# B&R Automation Studio project 305841_E00002_AM_0
Automation Studio 4.11.2.75; technology packages: mapp 5.17.0, mappCockpit 5.17.0, mappControl 5.17.0, mappMotion 5.17.1, mappSafety 5.17.0, mappView 5.17.0

## Configuration EchCm_AM

### Task classes (Cpu.sw)
```
Cyclic#2 (cycle 6000 us, tolerance 6000 us):
  ProdCycle <- PlcLogic.ProdCycle.prg
  Annunc <- PlcLogic.Annunc.prg
Cyclic#3 (cycle 12000 us, tolerance 12000 us):
  Pendant <- PlcLogic.Pendant.prg
  ProcInputs <- PlcLogic.ProcInputs.prg
  axSpinSM <- PlcLogic.axSpindle.axSpindleSM.prg
  axOutESM <- PlcLogic.axOutE.axOutESM.prg
  axInESM <- PlcLogic.axInE.axInESM.prg
  axZSM <- PlcLogic.axZ.axZSM.prg
  axHwSM <- PlcLogic.axHandwheel.axHwSM.prg
  axCfVfdSM <- PlcLogic.axCfVfd.axCfVfdSM.prg
Cyclic#4 (cycle 48000 us, tolerance 48000 us):
  AxEnable <- PlcLogic.AxEnable.prg
  CuttingFlu <- PlcLogic.CuttingFluidVFD.prg
  OmSafeDev <- PlcLogic.OmSafeDev.prg
  DepthToAng <- PlcLogic.DepthLookup.DepthToAngle.prg
DataObjects: McAcpSys
NcDataObjects: axSpindleP <- PlcLogic.axSpindle.axSpindleParamTable.dob, axOutEPara <- PlcLogic.axOutE.axOutEParamTable.dob, axInEParam <- PlcLogic.axInE.axInEParamTable.dob, axZParamTa <- PlcLogic.axZ.axZParamTable.dob, Cam1P <- PlcLogic.axInE.Cam1P.dob, Cam1P_Fp <- PlcLogic.axInE.Cam1P_Fp.dob, Cam2P <- PlcLogic.axInE.Cam2P.dob, Cam2P_Fp <- PlcLogic.axInE.Cam2P_Fp.dob, Cam3P <- PlcLogic.axInE.Cam3P.dob, Cam3P_Fp <- PlcLogic.axInE.Cam3P_Fp.dob, Cam4P <- PlcLogic.axInE.Cam4P.dob, Cam4P_Fp <- PlcLogic.axInE.Cam4P_Fp.dob, Cam5P <- PlcLogic.axInE.Cam5P.dob, Cam5P_Fp <- PlcLogic.axInE.Cam5P_Fp.dob, Cam6P <- PlcLogic.axInE.Cam6P.dob, Cam6P_Fp <- PlcLogic.axInE.Cam6P_Fp.dob, McDriveLog
Binaries: udbdef, mvLoader, arflatprv, TCData, FWRules, arcoal, arsvcreg, McAcpSim, McProfGen, McAcpDrv, mCoWebSc, TCLang, OpcUaSrv, DataObject, Settings, iomap, asfw, axCfgZ, Role, ashwac, sysconf, arconfig, ashwd, Config, axCfgInE, axCfgSpin, asiol1, axCfgOutE, Anonymous, User, cockpit1, TC, vAxHwCfg, vAxHw, axCfgCfPmp, CamFeature, camlist1, mappConfig, vAxHwLin, vAxHwRot, wgRecipe, cmRecipe, HwLinCfg, Config_5, HwRotCfg, Config_3
Libraries: sys_lib, runtime, brsystem, GAProcIO, standard, McBase, SfDomain, MpAxis, McAxis, MpBase, MpRecipe, McAcpAx, GAMpMotion, McPureVAx, astime, AsBrStr, GAConvert, MpAlarmX, AsBrMath, GAMath, CoTrace, AsZip, FileIO, McDS402Ax, astcp, asieccon, asiodiag, asepl, SfDomDrv, asusb, SfDomVis, aruser, arssl, powerlnk, MpSfDomMgr, dataobj, asioacc, GAMotor, MTFilter, MTBasics, MTTypes
```

### Hardware
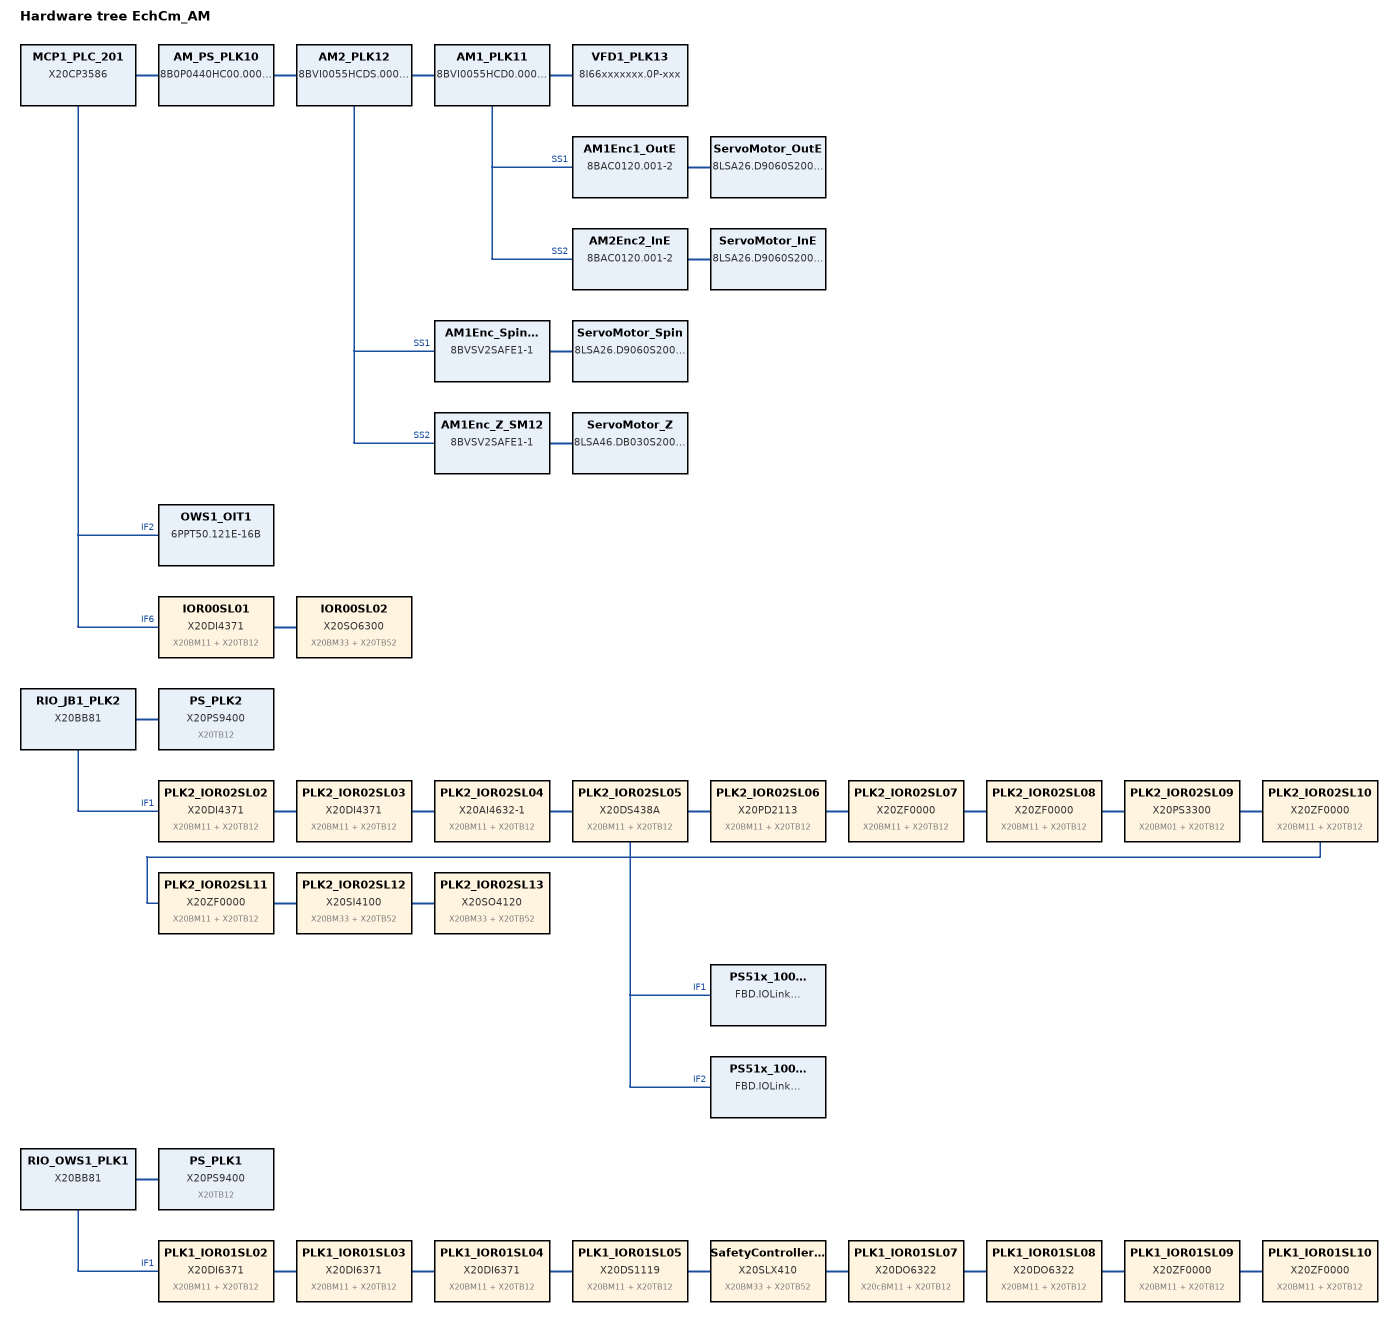
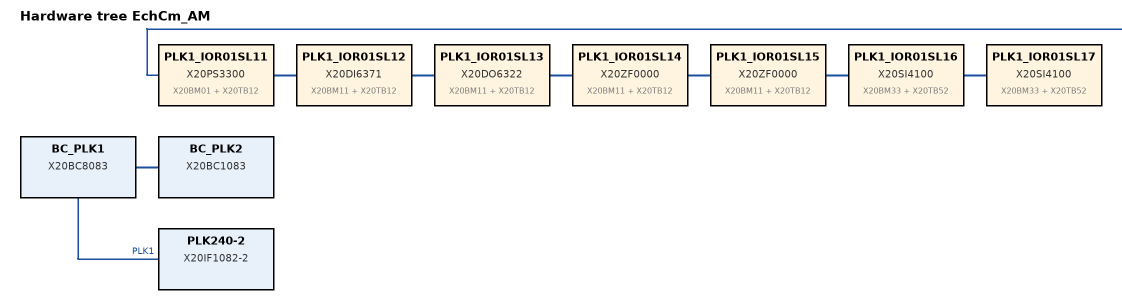
```
AM1Enc1_OutE : 8BAC0120.001-2 v2.2.0.0  [SS -> AM1_PLK11.SS1]
  PlugInType = Encoder
  McAcoposTypeID = AcoposMultiPlugInConfig
AM1Enc_Spin_SM11 : 8BVSV2SAFE1-1 v2.2.0.0  [SS -> AM2_PLK12.SS1]
  SafeModuleID = 11
  PlugInType = Encoder
  McAcoposTypeID = AcoposMultiPlugInConfig
AM1Enc_Z_SM12 : 8BVSV2SAFE1-1 v2.2.0.0  [SS -> AM2_PLK12.SS2]
  SafeModuleID = 12
  PlugInType = Encoder
  McAcoposTypeID = AcoposMultiPlugInConfig
AM1_PLK11 : 8BVI0055HCD0.000-1 v2.3.0.1  [PLK1 -> AM2_PLK12.PLK2 (NodeNumber=11) [Cable Type=PowerlinkCable, Length=10, Version=1.0.0.3]; PLK2 -> VFD1_PLK13.PLK1 (NodeNumber=11) [Cable Type=PowerlinkCable, Length=10, Version=1.0.0.3]; MT2 -> ServoMotor_InE.MT]
  DriveConfiguration/Module:
    McAcoposTypeID = AcoposP3SConfig
    ActivateACOPOSSimulationOnPLC = 0
  DriveConfiguration/Module/PowerSupply:
    PowerSupplyModuleReference = AM_PS
  DriveConfiguration/Channel[1]/RealAxis:
    AxisReference = gAxOutE
    MechanicalElementsIsInvisible = 0
  DriveConfiguration/Channel[1]/RealAxis/MechanicalElements/Gearbox:
    InputIsReadOnly = 0
    Input = 25
    OutputIsReadOnly = 0
    Output = 1
  DriveConfiguration/Channel[1]/RealAxis/MechanicalElements/RotaryToLinearTransformation:
    ReferenceDistanceIsReadOnly = 0
    ReferenceDistance = 360.0
  DriveConfiguration/Channel[1]/RealAxis/Controller:
    ModeIsReadOnly = 0
    Mode = PositionController
  DriveConfiguration/Channel[1]/RealAxis/Controller/Mode/Position:
    ProportionalGain = 462
    IntegrationTime = 0.0
    PredictionTime = 0.0004
    TotalDelayTime = 0.0004
  DriveConfiguration/Channel[1]/RealAxis/Controller/Mode/Speed:
    ProportionalGainIsReadOnly = 0
    ProportionalGain = 0.35
    IntegrationTimeIsReadOnly = 0
    IntegrationTime = 0.0
    FilterTimeIsReadOnly = 0
    FilterTime = 0.0
  DriveConfiguration/Channel[1]/RealAxis/Controller/Mode/LoopFilters:
    LoopFilterXIsReadOnly = 0
    LoopFilter1 = NotUsed
    LoopFilter2 = NotUsed
    LoopFilter3 = NotUsed
  DriveConfiguration/Channel[1]/RealAxis/Homing:
    ModeIsReadOnly = 0
    Mode = RestorePosition
    RestorePositionVariable = ::gr_AxOutERestorePos
  DriveConfiguration/Channel[1]/RealAxis/StopReaction:
    QuickstopIsReadOnly = 0
    Quickstop = DecelerationLimit
    DriveErrorIsReadOnly = 0
    DriveError = DecelerationLimit
  DriveConfiguration/Channel[1]/RealAxis/MovementErrorLimits:
    PositionError = 1.0
    VelocityErrorMonitoring = Automatic1
  DriveConfiguration/Channel[1]/RealAxis:
    JerkFilterIsReadOnly = 0
    JerkFilter = NotUsed
  DriveConfiguration/Channel[1]/RealAxis/DigitalInputs/HomingSwitch:
    SourceIsReadOnly = 0
    Source = NotUsed
    Level = High
  DriveConfiguration/Channel[1]/RealAxis/DigitalInputs/PositiveLimitSwitch:
    SourceIsReadOnly = 0
    Source = NotUsed
    Level = High
  DriveConfiguration/Channel[1]/RealAxis/DigitalInputs/NegativeLimitSwitch:
    SourceIsReadOnly = 0
    Source = NotUsed
    Level = High
  DriveConfiguration/Channel[1]/RealAxis/DigitalInputs/Trigger1:
    Source = X2Trigger1
    Level = High
  DriveConfiguration/Channel[1]/RealAxis/DigitalInputs/Trigger2:
    Source = X2Trigger2
    Level = High
  DriveConfiguration/Channel[1]/RealAxis/DigitalInputs/Quickstop:
    Input = NotUsed
  DriveConfiguration/Channel[1]/RealAxis/Simulation:
    SimulationModeOnPLC = SetValueGeneration
    SimulationModeOnACOPOS = NotUsed
  DriveConfiguration/Channel[1]:
    ExternalEncoderAxis = NotUsed
  DriveConfiguration/Channel[2]/RealAxis:
    AxisReference = gAxInE
    MechanicalElementsIsInvisible = 0
  DriveConfiguration/Channel[2]/RealAxis/MechanicalElements/Gearbox:
    InputIsReadOnly = 0
    Input = 25
    OutputIsReadOnly = 0
    Output = 1
  DriveConfiguration/Channel[2]/RealAxis/MechanicalElements/RotaryToLinearTransformation:
    ReferenceDistanceIsReadOnly = 0
    ReferenceDistance = 360.0
  DriveConfiguration/Channel[2]/RealAxis/Controller:
    ModeIsReadOnly = 0
    Mode = PositionController
  DriveConfiguration/Channel[2]/RealAxis/Controller/Mode/Position:
    ProportionalGain = 451.5
    IntegrationTime = 0.0
    PredictionTime = 0.0004
    TotalDelayTime = 0.0004
  DriveConfiguration/Channel[2]/RealAxis/Controller/Mode/Speed:
    ProportionalGainIsReadOnly = 0
    ProportionalGain = 0.325
    IntegrationTimeIsReadOnly = 0
    IntegrationTime = 0.0
    FilterTimeIsReadOnly = 0
    FilterTime = 0.0
  DriveConfiguration/Channel[2]/RealAxis/Controller/Mode/LoopFilters:
    LoopFilterXIsReadOnly = 0
    LoopFilter1 = NotUsed
    LoopFilter2 = NotUsed
    LoopFilter3 = NotUsed
  DriveConfiguration/Channel[2]/RealAxis/Homing:
    ModeIsReadOnly = 0
    Mode = RestorePosition
    RestorePositionVariable = ::gr_AxInERestorePos
  DriveConfiguration/Channel[2]/RealAxis/StopReaction:
    QuickstopIsReadOnly = 0
    Quickstop = DecelerationLimit
    DriveErrorIsReadOnly = 0
    DriveError = DecelerationLimit
  DriveConfiguration/Channel[2]/RealAxis/MovementErrorLimits:
    PositionError = 0.9
    VelocityErrorMonitoring = Automatic1
  DriveConfiguration/Channel[2]/RealAxis:
    JerkFilterIsReadOnly = 0
    JerkFilter = NotUsed
  DriveConfiguration/Channel[2]/RealAxis/DigitalInputs/HomingSwitch:
    SourceIsReadOnly = 0
    Source = NotUsed
    Level = High
  DriveConfiguration/Channel[2]/RealAxis/DigitalInputs/PositiveLimitSwitch:
    SourceIsReadOnly = 0
    Source = NotUsed
    Level = Low
  DriveConfiguration/Channel[2]/RealAxis/DigitalInputs/NegativeLimitSwitch:
    SourceIsReadOnly = 0
    Source = NotUsed
    Level = Low
  DriveConfiguration/Channel[2]/RealAxis/DigitalInputs/Trigger1:
    Source = X2Trigger1
    Level = High
  DriveConfiguration/Channel[2]/RealAxis/DigitalInputs/Trigger2:
    Source = X2Trigger2
    Level = High
  DriveConfiguration/Channel[2]/RealAxis/DigitalInputs/Quickstop:
    Input = NotUsed
  DriveConfiguration/Channel[2]/RealAxis/Simulation:
    SimulationModeOnPLC = SetValueGeneration
    SimulationModeOnACOPOS = NotUsed
  DriveConfiguration/Channel[2]/RealAxis/AxisFeatures:
    FeatureRef[1] = 
  DriveConfiguration/Channel[2]:
    ExternalEncoderAxis = NotUsed
  DriveConfiguration/Channel[2]/ChannelFeatures:
    FeatureRef[1] = Feature_CamList
AM2Enc2_InE : 8BAC0120.001-2 v2.2.0.0  [SS -> AM1_PLK11.SS2]
  PlugInType = Encoder
  McAcoposTypeID = AcoposMultiPlugInConfig
AM2_PLK12 : 8BVI0055HCDS.000-1 v2.3.0.1  [PLK1 -> AM_PS_PLK10.PLK2 (NodeNumber=12) [Cable Type=PowerlinkCable, Length=10, Version=1.0.0.3]; PLK2 -> AM1_PLK11.PLK1 (NodeNumber=12) [Cable Type=PowerlinkCable, Length=10, Version=1.0.0.3]; MT2 -> ServoMotor_Z.MT]
  DriveConfiguration/Module:
    McAcoposTypeID = AcoposMultiDConfig
    ActivateACOPOSSimulationOnPLC = 0
  DriveConfiguration/Module/PowerSupply:
    PowerSupplyModuleReference = AM_PS
  DriveConfiguration/Channel[1]/RealAxis:
    AxisReference = gAxSpin
    MechanicalElementsIsInvisible = 0
  DriveConfiguration/Channel[1]/RealAxis/MechanicalElements/Gearbox:
    InputIsReadOnly = 0
    Input = 10
    OutputIsReadOnly = 0
    Output = 1
  DriveConfiguration/Channel[1]/RealAxis/MechanicalElements/RotaryToLinearTransformation:
    ReferenceDistanceIsReadOnly = 0
    ReferenceDistance = 1
  DriveConfiguration/Channel[1]/RealAxis/Controller:
    ModeIsReadOnly = 0
    Mode = PositionController
  DriveConfiguration/Channel[1]/RealAxis/Controller/Mode/Position:
    ProportionalGain = 526
    IntegrationTime = 0.0
    PredictionTime = 0.0004
    TotalDelayTime = 0.0004
  DriveConfiguration/Channel[1]/RealAxis/Controller/Mode/Speed:
    ProportionalGainIsReadOnly = 0
    ProportionalGain = 0.25
    IntegrationTimeIsReadOnly = 0
    IntegrationTime = 0
    FilterTimeIsReadOnly = 0
    FilterTime = 0
  DriveConfiguration/Channel[1]/RealAxis/Controller/Mode/LoopFilters:
    LoopFilterXIsReadOnly = 0
    LoopFilter1 = NotUsed
    LoopFilter2 = NotUsed
    LoopFilter3 = NotUsed
  DriveConfiguration/Channel[1]/RealAxis/Homing:
    ModeIsReadOnly = 0
    Mode = RestorePosition
    RestorePositionVariable = ::gr_AxSpinRestorePos
  DriveConfiguration/Channel[1]/RealAxis/StopReaction:
    QuickstopIsReadOnly = 0
    Quickstop = DecelerationLimit
    DriveErrorIsReadOnly = 0
    DriveError = DecelerationLimit
  DriveConfiguration/Channel[1]/RealAxis/MovementErrorLimits:
    PositionError = 1.0
    VelocityErrorMonitoring = Automatic1
  DriveConfiguration/Channel[1]/RealAxis:
    JerkFilterIsReadOnly = 0
    JerkFilter = NotUsed
  DriveConfiguration/Channel[1]/RealAxis/DigitalInputs/HomingSwitch:
    SourceIsReadOnly = 0
    Source = NotUsed
    Level = High
  DriveConfiguration/Channel[1]/RealAxis/DigitalInputs/PositiveLimitSwitch:
    SourceIsReadOnly = 0
    Source = NotUsed
    Level = High
  DriveConfiguration/Channel[1]/RealAxis/DigitalInputs/NegativeLimitSwitch:
    SourceIsReadOnly = 0
    Source = NotUsed
    Level = High
  DriveConfiguration/Channel[1]/RealAxis/DigitalInputs/Trigger1:
    Source = X2Trigger1
    Level = High
  DriveConfiguration/Channel[1]/RealAxis/DigitalInputs/Trigger2:
    Source = X2Trigger2
    Level = High
  DriveConfiguration/Channel[1]/RealAxis/DigitalInputs/Quickstop:
    Input = NotUsed
  DriveConfiguration/Channel[1]/RealAxis/Simulation:
    SimulationModeOnPLC = SetValueGeneration
    SimulationModeOnACOPOS = NotUsed
  DriveConfiguration/Channel[1]:
    ExternalEncoderAxis = NotUsed
  DriveConfiguration/Channel[2]/RealAxis:
    AxisReference = gAxZ
    MechanicalElementsIsInvisible = 0
  DriveConfiguration/Channel[2]/RealAxis/MechanicalElements/Gearbox:
    InputIsReadOnly = 0
    Input = 1
    OutputIsReadOnly = 0
    Output = 1
  DriveConfiguration/Channel[2]/RealAxis/MechanicalElements/RotaryToLinearTransformation:
    ReferenceDistanceIsReadOnly = 0
    ReferenceDistance = 5.08
  DriveConfiguration/Channel[2]/RealAxis/Controller:
    ModeIsReadOnly = 0
    Mode = PositionController
  DriveConfiguration/Channel[2]/RealAxis/Controller/Mode/Position:
    ProportionalGain = 551
    IntegrationTime = 0.0
    PredictionTime = 0.0004
    TotalDelayTime = 0.0004
  DriveConfiguration/Channel[2]/RealAxis/Controller/Mode/Speed:
    ProportionalGainIsReadOnly = 0
    ProportionalGain = 1.0
    IntegrationTimeIsReadOnly = 0
    IntegrationTime = 0.0
    FilterTimeIsReadOnly = 0
    FilterTime = 0.0
  DriveConfiguration/Channel[2]/RealAxis/Controller/Mode/LoopFilters:
    LoopFilterXIsReadOnly = 0
    LoopFilter1 = NotUsed
    LoopFilter2 = NotUsed
    LoopFilter3 = NotUsed
  DriveConfiguration/Channel[2]/RealAxis/Homing:
    ModeIsReadOnly = 0
    Mode = RestorePosition
    RestorePositionVariable = ::gr_AxZRestorePos
  DriveConfiguration/Channel[2]/RealAxis/StopReaction:
    QuickstopIsReadOnly = 0
    Quickstop = DecelerationLimit
    DriveErrorIsReadOnly = 0
    DriveError = DecelerationLimit
  DriveConfiguration/Channel[2]/RealAxis/MovementErrorLimits:
    PositionError = 1.0
    VelocityErrorMonitoring = Automatic1
  DriveConfiguration/Channel[2]/RealAxis:
    JerkFilterIsReadOnly = 0
    JerkFilter = NotUsed
  DriveConfiguration/Channel[2]/RealAxis/DigitalInputs/HomingSwitch:
    SourceIsReadOnly = 0
    Source = NotUsed
    Level = High
  DriveConfiguration/Channel[2]/RealAxis/DigitalInputs/PositiveLimitSwitch:
    SourceIsReadOnly = 0
    Source = X2Trigger1
    Level = Low
  DriveConfiguration/Channel[2]/RealAxis/DigitalInputs/NegativeLimitSwitch:
    SourceIsReadOnly = 0
    Source = X2Trigger2
    Level = Low
  DriveConfiguration/Channel[2]/RealAxis/DigitalInputs/Trigger1:
    Source = X2Trigger1
    Level = High
  DriveConfiguration/Channel[2]/RealAxis/DigitalInputs/Trigger2:
    Source = X2Trigger2
    Level = High
  DriveConfiguration/Channel[2]/RealAxis/DigitalInputs/Quickstop:
    Input = NotUsed
  DriveConfiguration/Channel[2]/RealAxis/Simulation:
    SimulationModeOnPLC = SetValueGeneration
    SimulationModeOnACOPOS = NotUsed
  DriveConfiguration/Channel[2]/RealAxis/AxisFeatures:
    FeatureRef[1] = 
  DriveConfiguration/Channel[2]:
    ExternalEncoderAxis = NotUsed
AM_PS_PLK10 : 8B0P0440HC00.000-1 v2.3.0.1  [PLK1 -> MCP1_PLC_201.IF3 (NodeNumber=10) [Cable Type=PowerlinkCable, Length=10, Version=1.0.0.3]; PLK2 -> AM2_PLK12.PLK1 (NodeNumber=10) [Cable Type=PowerlinkCable, Length=10, Version=1.0.0.3]]
  DriveConfiguration/Module:
    McAcoposTypeID = AcoposMultiPSMpConfig
    ActivateACOPOSSimulationOnPLC = 0
  DriveConfiguration/Channel[1]/PowerSection:
    AxisReference = AM_PS
BC_PLK1 : X20BC8083 v2.14.0.0  [PLK1 -> PLK240-2.PLK2 (NodeNumber=1) [Cable Type=PowerlinkCable, Length=10, Version=1.0.0.3]; PLK2 -> BC_PLK2.PLK1 (NodeNumber=1) [Cable Type=PowerlinkCable, Length=10, Version=1.0.0.3]; SL -> RIO_OWS1_PLK1.SL1]
BC_PLK2 : X20BC1083 v2.14.0.0  [PLK1 -> BC_PLK1.PLK2 (NodeNumber=2) [Cable Type=PowerlinkCable, Length=10, Version=1.0.0.3]; SL -> RIO_JB1_PLK2.SL1]
IOR00SL01 : X20DI4371 v1.2.0.0  [SS1 -> X20TB12.SS; SL -> X20BM11.SL1]
IOR00SL02 : X20SO6300 v2.3.0.0  [SS1 -> X20TB52d.SS; SL -> X20BM33d.SL1]
  DigitalOutput01 = viaSafeLOGIC
  DigitalOutput02 = viaSafeLOGIC
  DigitalOutput03 = viaSafeLOGIC
  DigitalOutput04 = viaSafeLOGIC
  DigitalOutput05 = viaSafeLOGIC
  DigitalOutput06 = viaSafeLOGIC
MCP1_PLC_201 : X20CP3586 v1.10.0.0
  Connector IF2:
    ActivateDevice = 1
    HostName = plc_mcp1
    Mode = Manual
    InternetAddress = 10.10.2.240
    SubnetMask = 255.255.255.0
  Connector IF3:
    EplHostName = PLC_MCP1_PLK1
    CycleTime = 800
  ConfigurationID = 305841_E00002_Rev0_PLC_Main
  ConfigVersion = 0.0.0
  UserPartitionSize = 20
  AutomaticTransferOfUserfiles = on
  PermanentPvSize = 9216
  VolatileGlobalPvSize = 69630
  CyclicTaskClassCount = 6
  Cyclic1Duration = 2000
  Cyclic1Tolerance = 2000
  Cyclic2Duration = 6000
  Cyclic2Tolerance = 6000
  Cyclic3Duration = 12000
  Cyclic3Tolerance = 12000
  Cyclic4Duration = 48000
  Cyclic4Tolerance = 48000
  Cyclic5Duration = 96000
  Cyclic5Tolerance = 9600000
  Cyclic6Duration = 480000
  Cyclic6Tolerance = 480000
  FileDevice1
  FileDeviceName1 = UserPartitionRoot
  FileDevicePath1 = F:\
  FileDevice2
  FileDeviceName2 = Recipes
  FileDevicePath2 = F:\config\recipes\
  FileDevice3
  FileDeviceName3 = IOConfig
  FileDevicePath3 = F:\config\io\
  EthernetHostName = mcp1_plc201
  FtpUser1
  FtpUsername1 = ftpuser
  FtpUserPassword1 = wzi3iB5UNI3uCms7ZCmB0Woh2QaOICjzuPm+LM5DkNg=
  FtpUserSalt1 = UFkRbDjT
  FTPAccessRight1 = 0
  ActivateOpcUa = 1
  OpcUaPort = 4841
  OpcUaInformationModels_PV_Version = 1
OWS1_OIT1 : 6PPT50.121E-16B v1.3.8.0  [ETH1 -> MCP1_PLC_201.IF2 [Cable Type=PowerlinkCable, Length=10, Version=1.0.0.3]]
  Terminal = true
  Mode = Manual
  InternetAddress = 10.10.2.20
  Subnetmask = 255.255.255.0
  Hostname = ows1_oit1
  PasswordVNC = 
  PasswordCIFS = 
  PasswordService = 
PLK1_IOR01SL02 : X20DI6371 v1.2.0.0  [SS1 -> X20TB12n.SS; SL -> X20BM11l.SL1]
  InputFilter = 250
PLK1_IOR01SL03 : X20DI6371 v1.2.0.0  [SS1 -> X20TB12c.SS; SL -> X20BM11c.SL1]
  InputFilter = 250
PLK1_IOR01SL04 : X20DI6371 v1.2.0.0  [SS1 -> X20TB12ab.SS; SL -> X20BM11x.SL1]
  InputFilter = 250
PLK1_IOR01SL05 : X20DS1119 v1.5.0.0  [SS1 -> X20TB12e.SS; SL -> X20BM11e.SL1]
  PSInfo = on
  SDCInfo = on
  NetworkInfo = 8Bit
  Function03 = AB
PLK1_IOR01SL07 : X20DO6322 v1.3.0.0  [SS1 -> X20TB12p.SS; SL -> X20cBM11a.SL1]
PLK1_IOR01SL08 : X20DO6322 v1.3.0.0  [SS1 -> X20TB12h.SS; SL -> X20BM11h.SL1]
PLK1_IOR01SL09 : X20ZF0000 v1.1.0.0 (Disabled=true)  [SS1 -> X20TB12o.SS; SL -> X20BM11n.SL1]
PLK1_IOR01SL10 : X20ZF0000 v1.1.0.0 (Disabled=true)  [SS1 -> X20TB12i.SS; SL -> X20BM11m.SL1]
PLK1_IOR01SL11 : X20PS3300 v1.4.0.0  [SS1 -> X20TB12z.SS; SL -> X20BM01.SL1]
  PowerInfo = on
PLK1_IOR01SL12 : X20DI6371 v1.2.0.0  [SS1 -> X20TB12d.SS; SL -> X20BM11d.SL1]
PLK1_IOR01SL13 : X20DO6322 v1.3.0.0  [SS1 -> X20TB12b.SS; SL -> X20BM11b.SL1]
  Supervision = off
PLK1_IOR01SL14 : X20ZF0000 v1.1.0.0 (Disabled=true)  [SS1 -> X20TB12f.SS; SL -> X20BM11f.SL1]
PLK1_IOR01SL15 : X20ZF0000 v1.1.0.0 (Disabled=true)  [SS1 -> X20TB12q.SS; SL -> X20BM11o.SL1]
PLK1_IOR01SL16 : X20SI4100 v2.4.0.0  [SS1 -> X20TB52b.SS; SL -> X20BM33b.SL1]
  SafeModuleID = 116
PLK1_IOR01SL17 : X20SI4100 v2.4.0.0  [SS1 -> X20TB52a.SS; SL -> X20BM33a.SL1]
  SafeModuleID = 117
PLK240-2 : X20IF1082-2 v1.14.0.0  [PLK2 -> BC_PLK1.PLK1 [Cable Type=PowerlinkCable, Length=10, Version=1.0.0.3]; SS -> MCP1_PLC_201.SS1]
  Connector IF1:
    EplHostName = PLC_MCP1_PLK2
    NodeDefinition = Software
    EplNatSubnet = 192.168.102.0
PLK2_IOR02SL02 : X20DI4371 v1.2.0.0  [SS1 -> X20TB12s.SS; SL -> X20BM11p.SL1]
PLK2_IOR02SL03 : X20DI4371 v1.2.0.0  [SS1 -> X20TB12t.SS; SL -> X20BM11q.SL1]
PLK2_IOR02SL04 : X20AI4632-1 v1.2.0.0  [SS1 -> X20TB12u.SS; SL -> X20BM11r.SL1]
  ChannelType01 = 0 to 22mA
  ChannelType02 = 0 to 22mA
  Channel03enable = off
  Channel04enable = off
PLK2_IOR02SL05 : X20DS438A v2.4.0.0  [SS1 -> X20TB12aa.SS; SL -> X20BM11w.SL1]
  DtmRef = FBD.BRIOLinkModuleDTM.DTMCore.X20DS438A
  DtmId = 7db43003-0ff5-4bbd-8923-86eacecae911
  CommDtmId = ab9d1316-8c35-4493-ab34-f7b1b8ca9169
  RequiresDTMBuild = true
  ConfigFile = Communication.dtm
  ConfigModule = asiol1
  OperatingMode01 = Operate
  PDI_Enable01 = variousTypes
  PDI_DataType01_1 = UINT
  OperatingMode02 = Operate
  PDI_Enable02 = variousTypes
  PDI_DataType02_1 = UINT
PLK2_IOR02SL06 : X20PD2113 v1.2.0.0  [SS1 -> X20TB12g.SS; SL -> X20BM11g.SL1]
PLK2_IOR02SL07 : X20ZF0000 v1.1.0.0 (Disabled=true)  [SS1 -> X20TB12x.SS; SL -> X20BM11t.SL1]
PLK2_IOR02SL08 : X20ZF0000 v1.1.0.0 (Disabled=true)  [SS1 -> X20TB12w.SS; SL -> X20BM11v.SL1]
PLK2_IOR02SL09 : X20PS3300 v1.4.0.0 (Disabled=true)  [SS1 -> X20TB12ac.SS; SL -> X20BM01a.SL1]
  PowerInfo = on
PLK2_IOR02SL10 : X20ZF0000 v1.1.0.0 (Disabled=true)  [SS1 -> X20TB12y.SS; SL -> X20BM11u.SL1]
PLK2_IOR02SL11 : X20ZF0000 v1.1.0.0 (Disabled=true)  [SS1 -> X20TB12v.SS; SL -> X20BM11s.SL1]
PLK2_IOR02SL12 : X20SI4100 v2.4.0.0  [SS1 -> X20TB52c.SS; SL -> X20BM33c.SL1]
  SafeModuleID = 212
PLK2_IOR02SL13 : X20SO4120 v2.3.0.0  [SS1 -> X20TB52e.SS; SL -> X20BM33e.SL1]
  PLCopenInfo = on
  SafeModuleID = 213
  DigitalOutput01 = viaSafeLOGIC
  DigitalOutput02 = viaSafeLOGIC
  DigitalOutput03 = viaSafeLOGIC
  DigitalOutput04 = viaSafeLOGIC
PS51x_100_LI2UPN8_IODD1_1 : FBD.IOLink.GenericDeviceDTM.DTMCore.PS51x-100-LI2UPN8 IODD1.1 v2.9 (OrderNumber=PS51x-100-LI2UPN8 IODD1.1)  [IO-Link1 -> PLK2_IOR02SL05.IF1]
  DtmId = 9f03f336-de2c-4174-a814-ce0739b6707c
PS51x_100_LI2UPN8_IODD1_1a : FBD.IOLink.GenericDeviceDTM.DTMCore.PS51x-100-LI2UPN8 IODD1.1 v2.9 (OrderNumber=PS51x-100-LI2UPN8 IODD1.1)  [IO-Link1 -> PLK2_IOR02SL05.IF2]
  DtmId = 948ae1a5-f93f-40dc-8e06-a46fa964d649
PS_PLK1 : X20PS9400 v1.8.0.0  [SS1 -> X20TB12m.SS; PS -> RIO_OWS1_PLK1.PS1]
  PowerInfo = on
PS_PLK2 : X20PS9400 v1.8.0.0  [SS1 -> X20TB12r.SS; PS -> RIO_JB1_PLK2.PS1]
RIO_JB1_PLK2 : X20BB81 v1.1.0.0
RIO_OWS1_PLK1 : X20BB81 v1.1.0.0
SafetyController_R01SL06 : X20SLX410 v2.4.1.1  [SS1 -> X20TB52.SS; SL -> X20BM33.SL1]
  UnsafeOutputBOOLs = 24
  UnsafeInputBOOLs = 24
  UnsafeInputUINTs = 4
ServoMotor_InE : 8LSA26.D9060S200-3 v2.2.0.1  [EC -> AM2Enc2_InE.EC; MT -> AM1_PLK11.MT2]
  M1/MotorParameters:
    MOTOR_AMB_TEMP_RATED = 40
ServoMotor_OutE : 8LSA26.D9060S200-3 v2.2.0.1  [EC -> AM1Enc1_OutE.EC; MT -> AM1_PLK11.MT1]
  M1/MotorParameters:
    MOTOR_AMB_TEMP_RATED = 40
ServoMotor_Spin : 8LSA26.D9060S200-3 v2.2.0.1  [EC -> AM1Enc_Spin_SM11.EC; MT -> AM2_PLK12.MT1]
  M1/MotorParameters:
    MOTOR_AMB_TEMP_RATED = 40
ServoMotor_Z : 8LSA46.DB030S200-3 v2.2.0.1  [EC -> AM1Enc_Z_SM12.EC; MT -> AM2_PLK12.MT2]
  M1/MotorParameters:
    MOTOR_AMB_TEMP_RATED = 40
VFD1_PLK13 : 8I66xxxxxxx.0P-xxx v2.5.1.0  [PLK1 -> AM1_PLK11.PLK2 (NodeNumber=13) [Cable Type=PowerlinkCable, Length=10, Version=1.0.0.3]]
  Supervision = off
  PlkDiagnosisAdd = on
  FunctionModel = MotionConfig
  McTypeID = McAcoposInverterP66P
  AxisReference = gAxCfPmp
  InputIsReadOnly = 0
  Input = 1
  OutputIsReadOnly = 0
  Output = 1
  ReferenceDistanceIsReadOnly = 0
  ReferenceDistance = 1
  UnitOfSetpoint = Rpm
  IOM_AIDP1 = HMIS
  IOM_AIDP2 = LFT
  IOM_AIDP3 = ETAD_u
  Mode_LI3 = Safety
  Sel_NameplateMask = 8Ix6T401100_IEC
  Cfg_NSP = 1175
  Cfg_FRS = 600
  Cfg_UNS = 480
  Cfg_COS = 73
X20BM01 : X20BM01 v2.1.0.0  [X2X1 -> X20BM11m.X2X2]
X20BM01a : X20BM01 v2.1.0.0 (Disabled=true)  [X2X1 -> X20BM11v.X2X2]
X20BM11 : X20BM11 v1.1.0.0  [X2X1 -> MCP1_PLC_201.IF6]
X20BM11b : X20BM11 v1.1.0.0  [X2X1 -> X20BM11d.X2X2]
X20BM11c : X20BM11 v1.1.0.0  [X2X1 -> X20BM11l.X2X2]
X20BM11d : X20BM11 v1.1.0.0  [X2X1 -> X20BM01.X2X2]
X20BM11e : X20BM11 v1.1.0.0  [X2X1 -> X20BM11x.X2X2]
X20BM11f : X20BM11 v1.1.0.0 (Disabled=true)  [X2X1 -> X20BM11b.X2X2]
X20BM11g : X20BM11 v1.1.0.0  [X2X1 -> X20BM11w.X2X2]
X20BM11h : X20BM11 v1.1.0.0  [X2X1 -> X20cBM11a.X2X2]
X20BM11l : X20BM11 v1.1.0.0  [X2X1 -> RIO_OWS1_PLK1.IF1]
X20BM11m : X20BM11 v1.1.0.0 (Disabled=true)  [X2X1 -> X20BM11n.X2X2]
X20BM11n : X20BM11 v1.1.0.0 (Disabled=true)  [X2X1 -> X20BM11h.X2X2]
X20BM11o : X20BM11 v1.1.0.0 (Disabled=true)  [X2X1 -> X20BM11f.X2X2]
X20BM11p : X20BM11 v1.1.0.0  [X2X1 -> RIO_JB1_PLK2.IF1]
X20BM11q : X20BM11 v1.1.0.0  [X2X1 -> X20BM11p.X2X2]
X20BM11r : X20BM11 v1.1.0.0  [X2X1 -> X20BM11q.X2X2]
X20BM11s : X20BM11 v1.1.0.0 (Disabled=true)  [X2X1 -> X20BM11u.X2X2]
X20BM11t : X20BM11 v1.1.0.0 (Disabled=true)  [X2X1 -> X20BM11g.X2X2]
X20BM11u : X20BM11 v1.1.0.0 (Disabled=true)  [X2X1 -> X20BM01a.X2X2]
X20BM11v : X20BM11 v1.1.0.0 (Disabled=true)  [X2X1 -> X20BM11t.X2X2]
X20BM11w : X20BM11 v1.1.0.0  [X2X1 -> X20BM11r.X2X2]
X20BM11x : X20BM11 v1.1.0.0  [X2X1 -> X20BM11c.X2X2]
X20BM33 : X20BM33 v1.0.0.6  [X2X1 -> X20BM11e.X2X2]
X20BM33a : X20BM33 v1.0.0.6  [X2X1 -> X20BM33b.X2X2]
X20BM33b : X20BM33 v1.0.0.6  [X2X1 -> X20BM11o.X2X2]
X20BM33c : X20BM33 v1.0.0.6  [X2X1 -> X20BM11s.X2X2]
X20BM33d : X20BM33 v1.0.0.6  [X2X1 -> X20BM11.X2X2]
X20BM33e : X20BM33 v1.0.0.6  [X2X1 -> X20BM33c.X2X2]
X20TB12 : X20TB12 v1.0.0.0
X20TB12aa : X20TB12 v1.0.0.0
X20TB12ab : X20TB12 v1.0.0.0
X20TB12ac : X20TB12 v1.0.0.0 (Disabled=true)
X20TB12b : X20TB12 v1.0.0.0
X20TB12c : X20TB12 v1.0.0.0
X20TB12d : X20TB12 v1.0.0.0
X20TB12e : X20TB12 v1.0.0.0
X20TB12f : X20TB12 v1.0.0.0 (Disabled=true)
X20TB12g : X20TB12 v1.0.0.0
X20TB12h : X20TB12 v1.0.0.0
X20TB12i : X20TB12 v1.0.0.0 (Disabled=true)
X20TB12m : X20TB12 v1.0.0.0
X20TB12n : X20TB12 v1.0.0.0
X20TB12o : X20TB12 v1.0.0.0 (Disabled=true)
X20TB12p : X20TB12 v1.0.0.0
X20TB12q : X20TB12 v1.0.0.0 (Disabled=true)
X20TB12r : X20TB12 v1.0.0.0
X20TB12s : X20TB12 v1.0.0.0
X20TB12t : X20TB12 v1.0.0.0
X20TB12u : X20TB12 v1.0.0.0
X20TB12v : X20TB12 v1.0.0.0 (Disabled=true)
X20TB12w : X20TB12 v1.0.0.0 (Disabled=true)
X20TB12x : X20TB12 v1.0.0.0 (Disabled=true)
X20TB12y : X20TB12 v1.0.0.0 (Disabled=true)
X20TB12z : X20TB12 v1.0.0.0
X20TB52 : X20TB52 v1.0.0.2
X20TB52a : X20TB52 v1.0.0.2
X20TB52b : X20TB52 v1.0.0.2
X20TB52c : X20TB52 v1.0.0.2
X20TB52d : X20TB52 v1.0.0.2
X20TB52e : X20TB52 v1.0.0.2
X20cBM11a : X20cBM11 v1.0.1.0  [X2X1 -> X20BM33.X2X2]
```

### Cpu.per - MCP1_PLC_201/Cpu.per
```iecst
VAR_CONFIG
	gr_AxSpindleRestorePos AT %M0; (* *)
	gr_AxOutERestorePos AT %M72; (* *)
	gr_AxInERestorePos AT %M144; (* *)
	gr_AxZRestorePos AT %M216; (* *)
	gr_AI_FT_CFFlow_Params AT %M288; (* *)
	gr_AI_LT_CFTankLevel_Params AT %M376; (* *)
	gr_AI_PT_CFFilterOutlet_Params AT %M464; (* *)
	gr_AI_PT_CFPumpOutlet_Params AT %M552; (* *)
	gr_AI_DP_CFFilter_Params AT %M640; (* *)
	gr_DI_JI_480VACOk_Params AT %M728; (* *)
	gr_DI_LSL_CFTank_Params AT %M760; (* *)
	gr_DI_ZS_CFTankLocator_Params AT %M792; (* *)
	gr_AxisPositionLimits AT %M824; (* *)
	gr_CfgCurrent AT %M968; (* *)
	gr_PartCurrent AT %M1152; (* *)
END_VAR
```

### IoMap.iom - MCP1_PLC_201/IoMap.iom
```iecst
VAR_CONFIG
	::AI_FT_CFFlow.InRawINT AT %IW."PLK2_IOR02SL04".AnalogInput01;
	::AI_FT_CFFlow.ChannelOk AT %IX."PLK2_IOR02SL04".Channel01OK INVERSE;
	::AI_LT_CFTankLevel.InRawINT AT %IW."PLK2_IOR02SL04".AnalogInput02;
	::AI_LT_CFTankLevel.ChannelOk AT %IX."PLK2_IOR02SL04".Channel02OK INVERSE;
	::ModStat_JB1_PLK2.Slot05ModuleOk AT %IX."PLK2_IOR02SL05".ModuleOk;
	::ModStat_JB1_PLK2.Slot02ModuleOk AT %IX."PLK2_IOR02SL02".ModuleOk;
	::ModStat_JB1_PLK2.Slot03ModuleOk AT %IX."PLK2_IOR02SL03".ModuleOk;
	::ModStat_JB1_PLK2.Slot04ModuleOk AT %IX."PLK2_IOR02SL04".ModuleOk;
	::ModStat_JB1_PLK2.Slot06ModuleOk AT %IX."PLK2_IOR02SL06".ModuleOk;
	::ModStat_JB1_PLK2.Slot09ModuleOk AT %IX."PLK2_IOR02SL09".ModuleOk;
	::ModStat_JB1_PLK2.Slot12ModuleOk AT %IX."PLK2_IOR02SL12".ModuleOk;
	::ModStat_JB1_PLK2.Slot13ModuleOk AT %IX."PLK2_IOR02SL13".ModuleOk;
	::ModStat_OWS_PLK1.Slot02ModuleOk AT %IX."PLK1_IOR01SL02".ModuleOk;
	::ModStat_OWS_PLK1.Slot03ModuleOk AT %IX."PLK1_IOR01SL03".ModuleOk;
	::ModStat_OWS_PLK1.Slot04ModuleOk AT %IX."PLK1_IOR01SL04".ModuleOk;
	::ModStat_OWS_PLK1.Slot05ModuleOk AT %IX."PLK1_IOR01SL05".ModuleOk;
	::ModStat_OWS_PLK1.Slot07ModuleOk AT %IX."PLK1_IOR01SL07".ModuleOk;
	::ModStat_OWS_PLK1.Slot08ModuleOk AT %IX."PLK1_IOR01SL08".ModuleOk;
	::ModStat_OWS_PLK1.Slot11ModuleOk AT %IX."PLK1_IOR01SL11".ModuleOk;
	::ModStat_OWS_PLK1.Slot12ModuleOk AT %IX."PLK1_IOR01SL12".ModuleOk;
	::ModStat_OWS_PLK1.Slot13ModuleOk AT %IX."PLK1_IOR01SL13".ModuleOk;
	::ModStat_OWS_PLK1.Slot16ModuleOk AT %IX."PLK1_IOR01SL16".ModuleOk;
	::ModStat_OWS_PLK1.Slot17ModuleOk AT %IX."PLK1_IOR01SL17".ModuleOk;
	::ModStat_PLC_201.Slot01ModuleOk AT %IX."IOR00SL01".ModuleOk;
	::ModStat_OWS_PLK1.Slot06ModuleOk AT %IX."SafetyController_R01SL06".ModuleOk;
	::DI_LSL_CFTank.InRaw AT %IX."PLK2_IOR02SL02".DigitalInput01;
	::DI_ZS_CFTankLocator.InRaw AT %IX."PLK2_IOR02SL02".DigitalInput02;
	::DI_JI_480VACOk.InRaw AT %IX."IOR00SL01".DigitalInput01;
	::owsPendant.AxisSelectInputs[1] AT %IX."PLK1_IOR01SL02".DigitalInput01;
	::owsPendant.AxisSelectInputs[2] AT %IX."PLK1_IOR01SL02".DigitalInput02;
	::owsPendant.AxisSelectInputs[3] AT %IX."PLK1_IOR01SL02".DigitalInput03;
	::owsPendant.SpeedSelectInputs[1] AT %IX."PLK1_IOR01SL02".DigitalInput04;
	::owsPendant.SpeedSelectInputs[2] AT %IX."PLK1_IOR01SL02".DigitalInput05;
	::owsPendant.SpeedSelectInputs[3] AT %IX."PLK1_IOR01SL02".DigitalInput06;
	::owsPendant.PBInputs[1] AT %IX."PLK1_IOR01SL03".DigitalInput01;
	::owsPendant.PBInputs[2] AT %IX."PLK1_IOR01SL03".DigitalInput02;
	::owsPendant.PBInputs[3] AT %IX."PLK1_IOR01SL03".DigitalInput03;
	::owsPendant.PBInputs[4] AT %IX."PLK1_IOR01SL03".DigitalInput04;
	::owsPendant.PBInputs[5] AT %IX."PLK1_IOR01SL03".DigitalInput05;
	::owsPendant.PBInputs[6] AT %IX."PLK1_IOR01SL03".DigitalInput06;
	::owsPendant.PBInputs[7] AT %IX."PLK1_IOR01SL04".DigitalInput01;
	::owsPendant.PBInputs[8] AT %IX."PLK1_IOR01SL04".DigitalInput02;
	::owsPendant.PBInputs[9] AT %IX."PLK1_IOR01SL04".DigitalInput03;
	::owsPendant.tmrCountResetPulse.Q AT %QX."PLK1_IOR01SL05".CounterReset;
	::owsPendant.encoderPowerOk AT %IX."PLK1_IOR01SL05".PowerSupply02 INVERSE;
	::owsPendant.HandwheelCounter AT %ID."PLK1_IOR01SL05".CounterValue01;
	::axes[1].Status.SafeMotionDiagCode AT %IW."SafetyController_R01SL06".UINT0001;
	::axes[2].Status.SafeMotionDiagCode AT %IW."SafetyController_R01SL06".UINT0002;
	::axes[3].Status.SafeMotionDiagCode AT %IW."SafetyController_R01SL06".UINT0003;
	::axes[4].Status.SafeMotionDiagCode AT %IW."SafetyController_R01SL06".UINT0004;
	::OmSafeDev:fs_EmoCmd AT %IX."SafetyController_R01SL06".BOOL00001;
	::OmSafeDev:fs_AllSMsOk AT %IX."SafetyController_R01SL06".BOOL00002;
	::OmSafeDev:fs_EmoOwsOk AT %IX."SafetyController_R01SL06".BOOL00007;
	::owsPendant.emoAcivated AT %IX."SafetyController_R01SL06".BOOL00008;
	::OmSafeDev:fs_StartPbOk AT %IX."SafetyController_R01SL06".BOOL00013;
	::OmSafeDev:fs_KeyswitchInRun AT %IX."SafetyController_R01SL06".BOOL00014;
	::OmSafeDev:fs_KeyswitchOk AT %IX."SafetyController_R01SL06".BOOL00015;
	::owsPendant.enableSwActive AT %IX."SafetyController_R01SL06".BOOL00017;
	::OmSafeDev:fs_CfGateClosed AT %IX."SafetyController_R01SL06".BOOL00019;
	::axes[4].Commands.ReleaseBrakeCmd AT %QX."SafetyController_R01SL06".BOOL10016;
	::axes[3].Commands.ReleaseBrakeCmd AT %QX."SafetyController_R01SL06".BOOL10015;
	::axes[2].Commands.ReleaseBrakeCmd AT %QX."SafetyController_R01SL06".BOOL10014;
	::axes[1].Commands.ReleaseBrakeCmd AT %QX."SafetyController_R01SL06".BOOL10013;
	::OmSafeDev:ts_ResetEStop AT %QX."SafetyController_R01SL06".BOOL10001;
	::OmSafeDev:ts_ResetSafeMC AT %QX."SafetyController_R01SL06".BOOL10002;
	::axes[1].Commands.PlcSafetyEnable AT %QX."SafetyController_R01SL06".BOOL10008;
	::axes[2].Commands.PlcSafetyEnable AT %QX."SafetyController_R01SL06".BOOL10009;
	::axes[3].Commands.PlcSafetyEnable AT %QX."SafetyController_R01SL06".BOOL10010;
	::axes[4].Commands.PlcSafetyEnable AT %QX."SafetyController_R01SL06".BOOL10011;
	::OmSafeDev:ts_InEmoMode AT %QX."SafetyController_R01SL06".BOOL10003;
	::OmSafeDev:ts_InSafeMode AT %QX."SafetyController_R01SL06".BOOL10004;
	::OmSafeDev:ts_InPendantMode AT %QX."SafetyController_R01SL06".BOOL10005;
	::OmSafeDev:fs_CfGateClosedLocked AT %IX."SafetyController_R01SL06".BOOL00020;
	::DO_PL_OWSGreen AT %QX."PLK1_IOR01SL13".DigitalOutput01;
	::DO_PL_OWSAmber AT %QX."PLK1_IOR01SL13".DigitalOutput02;
	::DO_PL_OWSRed AT %QX."PLK1_IOR01SL13".DigitalOutput03;
	::DO_PL_OWSBeconGreen AT %QX."PLK1_IOR01SL13".DigitalOutput04;
	::DO_PL_OWSBeconAmber AT %QX."PLK1_IOR01SL13".DigitalOutput05;
	::DO_PL_OWSBeconRed AT %QX."PLK1_IOR01SL13".DigitalOutput06;
	::ProcInputs:AI_PT_CFPumpOutletRaw AT %IW."PLK2_IOR02SL05".InputData01_1;
	::ProcInputs:AI_PT_CFFilterOutletRaw AT %IW."PLK2_IOR02SL05".InputData02_1;
	::owsPendant.emoWiringOk AT %IX."SafetyController_R01SL06".BOOL00009;
	::OmSafeDev:fs_StopPbActive AT %IX."SafetyController_R01SL06".BOOL00010;
	::owsPendant.pendantAllowMoves AT %IX."SafetyController_R01SL06".BOOL00003;
	::OmSafeDev:fs_EmoOwsActive AT %IX."SafetyController_R01SL06".BOOL00006;
	::OmSafeDev:fs_StopPbOk AT %IX."SafetyController_R01SL06".BOOL00011;
	::OmSafeDev:fs_StartPbActive AT %IX."SafetyController_R01SL06".BOOL00012;
	::owsPendant.enableSwWiringOk AT %IX."SafetyController_R01SL06".BOOL00018;
	::ProdCycle:ts_InCycle AT %QX."SafetyController_R01SL06".BOOL10006;
	::ProdCycle:ts_cfLockGate AT %QX."SafetyController_R01SL06".BOOL10007;
	::OmSafeDev:fs_InSafeMode AT %IX."SafetyController_R01SL06".BOOL00016;
	::ModStat_PLC_201.Slot02ModuleOk AT %IX."IOR00SL02".ModuleOk;
	::owsPendant.PLCmds[1] AT %QX."PLK1_IOR01SL07".DigitalOutput01;
	::owsPendant.PLCmds[2] AT %QX."PLK1_IOR01SL07".DigitalOutput02;
	::owsPendant.PLCmds[3] AT %QX."PLK1_IOR01SL07".DigitalOutput03;
	::owsPendant.PLCmds[4] AT %QX."PLK1_IOR01SL07".DigitalOutput04;
	::owsPendant.PLCmds[5] AT %QX."PLK1_IOR01SL07".DigitalOutput05;
	::owsPendant.PLCmds[6] AT %QX."PLK1_IOR01SL07".DigitalOutput06;
	::owsPendant.PLCmds[7] AT %QX."PLK1_IOR01SL08".DigitalOutput01;
	::owsPendant.PLCmds[8] AT %QX."PLK1_IOR01SL08".DigitalOutput02;
	::owsPendant.PLCmds[9] AT %QX."PLK1_IOR01SL08".DigitalOutput03;
	::DO_PB_OWSGreen AT %QX."PLK1_IOR01SL08".DigitalOutput04;
	::DO_PB_OWSRed AT %QX."PLK1_IOR01SL08".DigitalOutput05;
	::OmSafeDev:fs_CfGateClosedOk AT %IX."SafetyController_R01SL06".BOOL00021;
	::owsPendant.pendantPowerOk AT %IX."PLK1_IOR01SL05".PowerSupply01 INVERSE;
	::axes[8].Commands.PlcSafetyEnable AT %QX."SafetyController_R01SL06".BOOL10012;
	::OmSafeDev:ts_InManualMode AT %QX."SafetyController_R01SL06".BOOL10017;
	::OmSafeDev:ts_InProductionMode AT %QX."SafetyController_R01SL06".BOOL10018;
	::cfVfd.isModuleOk AT %IX."VFD1_PLK13".ModuleOk;
	::cfVfd.DevSpecStatus AT %IW."VFD1_PLK13".HMIS_Input;
	::cfVfd.DevSpecError AT %IW."VFD1_PLK13".LFT_Input;
	::cfVfd.StdError AT %IW."VFD1_PLK13".ErrorCode_I603F;
	::cfVfd.StdStatus AT %IW."VFD1_PLK13".StatusWord_I6041;
	::cfVfd.VelCommanded AT %IW."VFD1_PLK13".VlVelocityDemand_I6043;
	::cfVfd.VelAct AT %IW."VFD1_PLK13".VlVelocityActualValue_I6044;
END_VAR
```

### CamFeature.axisfeature - MCP1_PLC_201/mappMotion/Eccentrics/CamFeature.axisfeature
```
Element Feature_CamList (Type=axisfeature)
  Type = CamList
    CamListRef = CamList_1
```

### axCfgInE.axis - MCP1_PLC_201/mappMotion/Eccentrics/axCfgInE.axis
```
Element gAxInE (Type=axis)
  BaseTypeIsReadOnly = 0
  BaseType = RotaryPeriodic
    MeasurementUnitIsReadOnly = 0
    MeasurementUnit = 17476
    MeasurementResolutionIsReadOnly = 0
    MeasurementResolution = 0.001
    CountDirectionIsReadOnly = 0
    CountDirection = Standard
    PeriodSettings:
      Period = 360.0
  MovementLimitsIsReadOnly = 0
  MovementLimits = Internal
    Position:
      LowerLimitMin = -1.79769313486231E308
      UpperLimitMax = 1.79769313486231E308
      LowerLimit = -1000.0
      UpperLimit = 1000.0
    VelocityIsReadOnly = 0
    Velocity:
      VelocityMax = 3.4E38
      Velocity = 25
    AccelerationIsReadOnly = 0
    Acceleration:
      AccelerationMax = 3.4E38
      Acceleration = 25
    DecelerationIsReadOnly = 0
    Deceleration:
      DecelerationMax = 3.4E38
      Deceleration = 80
  Alarms = MpAlarmX
```

### axCfgOutE.axis - MCP1_PLC_201/mappMotion/Eccentrics/axCfgOutE.axis
```
Element gAxOutE (Type=axis)
  BaseTypeIsReadOnly = 0
  BaseType = RotaryPeriodic
    MeasurementUnitIsReadOnly = 0
    MeasurementUnit = 17476
    MeasurementResolutionIsReadOnly = 0
    MeasurementResolution = 0.001
    CountDirectionIsReadOnly = 0
    CountDirection = Standard
    PeriodSettings:
      Period = 360.0
  MovementLimitsIsReadOnly = 0
  MovementLimits = Internal
    Position:
      LowerLimitMin = -1.79769313486231E308
      UpperLimitMax = 1.79769313486231E308
      LowerLimit = -1000.0
      UpperLimit = 1000.0
    VelocityIsReadOnly = 0
    Velocity:
      VelocityMax = 3.4E38
      Velocity = 1600
    AccelerationIsReadOnly = 0
    Acceleration:
      AccelerationMax = 3.4E38
      Acceleration = 1600
    DecelerationIsReadOnly = 0
    Deceleration:
      DecelerationMax = 3.4E38
      Deceleration = 6000
  Alarms = MpAlarmX
```

### camlist1.camlist - MCP1_PLC_201/mappMotion/Eccentrics/camlist1.camlist
```
Element CamList_1 (Type=camlist)
  Row[1]:
    CamName = Cam1P
    CamID = 1
    Description
  Row[2]:
    CamName = CamBigP
    CamID = 2
    Description
```

### axCfgCfPmp.axis - MCP1_PLC_201/mappMotion/axCfgCfPmp.axis
```
Element gAxCfPmp (Type=axis)
  BaseTypeIsReadOnly = 0
  BaseType = Rotary
    MeasurementUnitIsReadOnly = 0
    MeasurementUnit = 5059636
    MeasurementResolutionIsReadOnly = 0
    MeasurementResolution = 1.0
    CountDirectionIsReadOnly = 0
    CountDirection = Standard
  MovementLimitsIsReadOnly = 0
  MovementLimits = Internal
    Position:
      LowerLimitMin = -1.79769313486231E308
      UpperLimitMax = 1.79769313486231E308
      LowerLimit = -1000.0
      UpperLimit = 1000.0
    VelocityIsReadOnly = 0
    Velocity:
      VelocityMax = 3.4E38
      Velocity = 24
    AccelerationIsReadOnly = 0
    Acceleration:
      AccelerationMax = 3.4E38
      Acceleration = 24
    DecelerationIsReadOnly = 0
    Deceleration:
      DecelerationMax = 3.4E38
      Deceleration = 24
  Alarms = MpAlarmX
```

### axCfgSpin.axis - MCP1_PLC_201/mappMotion/axCfgSpin.axis
```
Element gAxSpin (Type=axis)
  BaseTypeIsReadOnly = 0
  BaseType = RotaryPeriodic
    MeasurementUnitIsReadOnly = 0
    MeasurementUnit = 5059636
    MeasurementResolutionIsReadOnly = 0
    MeasurementResolution = 0.01
    CountDirectionIsReadOnly = 0
    CountDirection = Inverse
    PeriodSettings:
      Period = 1.0
  MovementLimitsIsReadOnly = 0
  MovementLimits = Internal
    Position:
      LowerLimitMin = -1.79769313486231E308
      UpperLimitMax = 1.79769313486231E308
      LowerLimit = -1000.0
      UpperLimit = 1000.0
    VelocityIsReadOnly = 0
    Velocity:
      VelocityMax = 3.4E38
      Velocity = 20
    AccelerationIsReadOnly = 0
    Acceleration:
      AccelerationMax = 3.4E38
      Acceleration = 20
    DecelerationIsReadOnly = 0
    Deceleration:
      DecelerationMax = 3.4E38
      Deceleration = 60
  Alarms = MpAlarmX
```

### axCfgZ.axis - MCP1_PLC_201/mappMotion/axCfgZ.axis
```
Element gAxZ (Type=axis)
  BaseTypeIsReadOnly = 0
  BaseType = LinearBounded
    MeasurementUnit = 5066068
    MeasurementResolutionIsReadOnly = 0
    MeasurementResolution = 0.001
    CountDirectionIsReadOnly = 0
    CountDirection = Inverse
  MovementLimitsIsReadOnly = 0
  MovementLimits = Internal
    Position:
      LowerLimitMin = -1.79769313486231E308
      UpperLimitMax = 1.79769313486231E308
      LowerLimit = 17
      UpperLimit = 3400
    VelocityIsReadOnly = 0
    Velocity:
      VelocityMax = 3.4E38
      Velocity = 125
    AccelerationIsReadOnly = 0
    Acceleration:
      AccelerationMax = 3.4E38
      Acceleration = 30
    DecelerationIsReadOnly = 0
    Deceleration:
      DecelerationMax = 3.4E38
      Deceleration = 250
  Alarms = MpAlarmX
```

### mappConfig.mappmotioncfg - MCP1_PLC_201/mappMotion/mappConfig.mappmotioncfg
```
Element MappMotionConfiguration (Type=mappmotioncfg)
  Processing:
    ProcessingTaskClass = 2
```

- Safety project (password-protected, skipped)

### angleLu.mprecipecsv - MCP1_PLC_201/mappServices/angleLu.mprecipecsv
```
Element angleLuRecipeCsv (Type=mprecipecsv)
  mapp.Recipe.Csv:
    Format:
      ColumnSeparator = ,
      DecimalMark = .
  Alarms = None
```

### depthLu.mprecipecsv - MCP1_PLC_201/mappServices/depthLu.mprecipecsv
```
Element depthLuRecipeCsv (Type=mprecipecsv)
  mapp.Recipe.Csv:
    Format:
      ColumnSeparator = ,
      DecimalMark = .
  Alarms = None
```

## Configuration EchCm_P3

CPU X20CP3586, AutomationRuntime B4.91, Build 6.3.0, Safety 0.0, Vc V4.72.5

### Task classes (Cpu.sw)
```
Cyclic#2 (cycle 6000 us, tolerance 6000 us):
  ProdCycle <- PlcLogic.ProdCycle.prg
  Annunc <- PlcLogic.Annunc.prg
Cyclic#3 (cycle 12000 us, tolerance 12000 us):
  Pendant <- PlcLogic.Pendant.prg
  ProcInputs <- PlcLogic.ProcInputs.prg
  axSpinSM <- PlcLogic.axSpindle.axSpindleSM.prg
  axOutESM <- PlcLogic.axOutE.axOutESM.prg
  axInESM <- PlcLogic.axInE.axInESM.prg
  axZSM <- PlcLogic.axZ.axZSM.prg
  axHwSM <- PlcLogic.axHandwheel.axHwSM.prg
  axCfVfdSM <- PlcLogic.axCfVfd.axCfVfdSM.prg
Cyclic#4 (cycle 48000 us, tolerance 48000 us):
  AxEnable <- PlcLogic.AxEnable.prg
  CuttingFlu <- PlcLogic.CuttingFluidVFD.prg
  OmSafeDev <- PlcLogic.OmSafeDev.prg
DataObjects: McAcpSys
NcDataObjects: axZParamTa <- PlcLogic.axZ.axZParamTable.dob, McDriveLog
Binaries: udbdef, mvLoader, arflatprv, TCData, FWRules, arcoal, arsvcreg, McAcpSim, McProfGen, McAcpDrv, mCoWebSc, TCLang, OpcUaSrv, DataObject, Settings, iomap, asfw, axCfgZ, Role, ashwac, sysconf, arconfig, ashwd, Config, axCfgInE, axCfgSpin, asiol1, axCfgOutE, Anonymous, User, cockpit1, TC, vAxHwCfg, vAxHw, axCfgCfPmp, vAxHwLin, vAxHwRot, wgRecipe, cmRecipe, HwLinCfg, Config_5, HwRotCfg, Config_3
Libraries: sys_lib, runtime, brsystem, GAProcIO, standard, McBase, SfDomain, MpAxis, McAxis, MpBase, MpRecipe, McAcpAx, GAMpMotion, McPureVAx, astime, AsBrStr, GAConvert, MpAlarmX, AsBrMath, GAMath, CoTrace, AsZip, FileIO, McDS402Ax, astcp, asieccon, asiodiag, asepl, SfDomDrv, asusb, SfDomVis, aruser, arssl, powerlnk, MpSfDomMgr, dataobj, asioacc, GAMotor, MTFilter, MTBasics, MTTypes
```

### Hardware
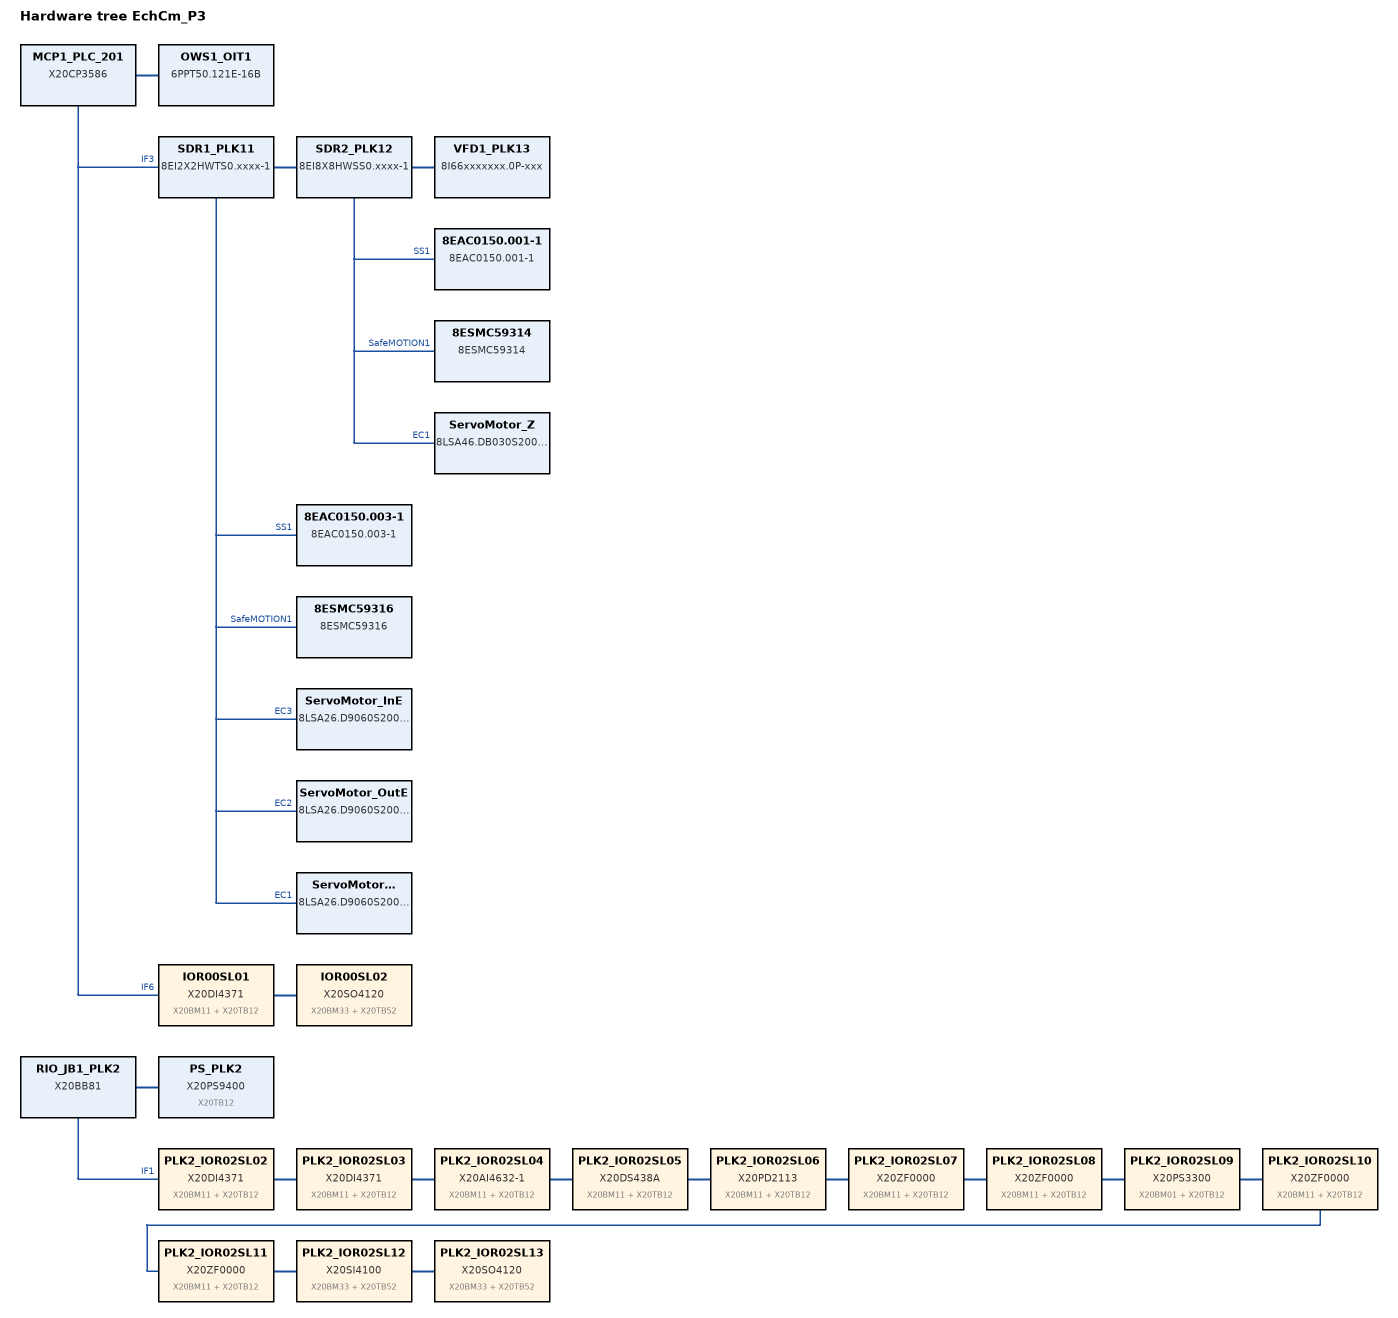
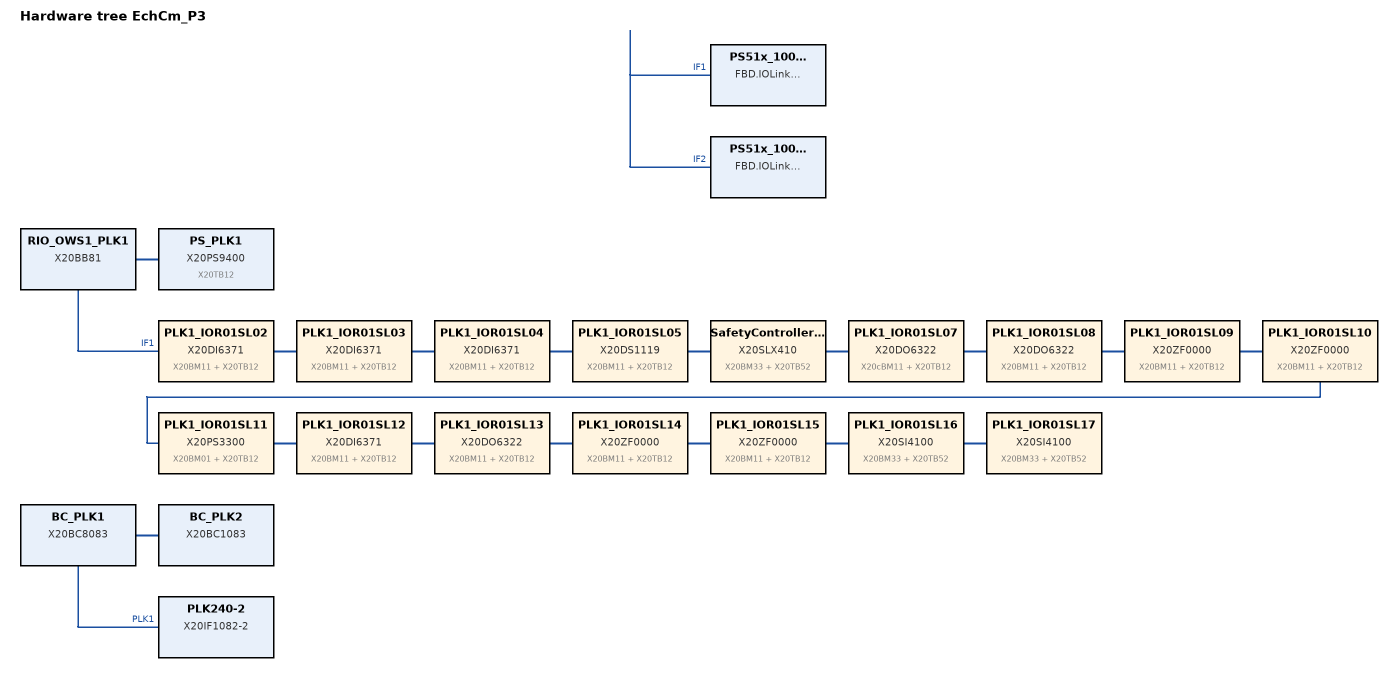
```
8EAC0150.001-1 : 8EAC0150.001-1 v2.2.0.4  [SS -> SDR2_PLK12.SS1]
  PlugInType = Encoder
  McAcoposTypeID = AcoposP3PlugInSConfig
  InterfaceType = EnDat
8EAC0150.003-1 : 8EAC0150.003-1 v2.2.0.4  [SS -> SDR1_PLK11.SS1]
  Encoder:
    PlugInType = Encoder
    McAcoposTypeID = AcoposP3PlugInTConfig
  Encoder/EncoderX42x:
    InterfaceType = NotUsed
  Encoder/EncoderX43x:
    InterfaceType = NotUsed
8ESMC59314 : 8ESMC59314 v2.2.0.0  [SafeMOTION -> SDR2_PLK12.SafeMOTION1]
  SafeModuleID = 12
8ESMC59316 : 8ESMC59316 v2.2.0.0  [SafeMOTION -> SDR1_PLK11.SafeMOTION1]
  SafeModuleID = 11
BC_PLK1 : X20BC8083 v2.11.1.0  [PLK1 -> PLK240-2.PLK2 (NodeNumber=1) [Cable Type=PowerlinkCable, Length=10, Version=1.0.0.3]; PLK2 -> BC_PLK2.PLK1 (NodeNumber=1) [Cable Type=PowerlinkCable, Length=10, Version=1.0.0.3]; SL -> RIO_OWS1_PLK1.SL1]
BC_PLK2 : X20BC1083 v2.12.0.0  [PLK1 -> BC_PLK1.PLK2 (NodeNumber=2) [Cable Type=PowerlinkCable, Length=10, Version=1.0.0.3]; SL -> RIO_JB1_PLK2.SL1]
IOR00SL01 : X20DI4371 v1.1.0.0  [SS1 -> X20TB12.SS; SL -> X20BM11.SL1]
IOR00SL02 : X20SO4120 v2.2.1.0  [SS1 -> X20TB52d.SS; SL -> X20BM33d.SL1]
  Supervision = off
  DigitalOutput01 = viaSafeLOGIC
  DigitalOutput02 = viaSafeLOGIC
  DigitalOutput03 = viaSafeLOGIC
  DigitalOutput04 = viaSafeLOGIC
MCP1_PLC_201 : X20CP3586 v1.9.0.0
  Connector IF2:
    ActivateDevice = 1
    HostName = plc_mcp1
    Mode = Manual
    InternetAddress = 10.10.2.240
    SubnetMask = 255.255.255.0
  Connector IF3:
    EplHostName = PLC_MCP1_PLK1
    CycleTime = 800
  ConfigurationID = 305841_E00002_Rev0_PLC_Main
  ConfigVersion = 0.0.0
  UserPartitionSize = 20
  Simulation = 1
  PermanentPvSize = 9216
  CyclicTaskClassCount = 6
  Cyclic1Duration = 2000
  Cyclic1Tolerance = 2000
  Cyclic2Duration = 6000
  Cyclic2Tolerance = 6000
  Cyclic3Duration = 12000
  Cyclic3Tolerance = 12000
  Cyclic4Duration = 48000
  Cyclic4Tolerance = 48000
  Cyclic5Duration = 96000
  Cyclic5Tolerance = 96000
  Cyclic6Duration = 480000
  Cyclic6Tolerance = 480000
  FileDevice1
  FileDeviceName1 = IOScaling
  FileDevicePath1 = F:\config\io\
  FileDevice2
  FileDeviceName2 = Recipes
  FileDevicePath2 = F:\config\recipes\
  EthernetHostName = mcp1_plc201
  ActivateOpcUa = 1
  OpcUaPort = 4841
  OpcUaInformationModels_PV_Version = 1
OWS1_OIT1 : 6PPT50.121E-16B v1.3.3.0  [ETH1 -> MCP1_PLC_201.IF2 [Cable Type=PowerlinkCable, Length=10, Version=1.0.0.3]]
  Terminal = true
  Mode = Manual
  InternetAddress = 10.10.2.20
  Subnetmask = 255.255.255.0
  Hostname = ows1_oit1
  PasswordVNC = 
  PasswordCIFS = 
  PasswordService = 
PLK1_IOR01SL02 : X20DI6371 v1.1.0.0  [SS1 -> X20TB12n.SS; SL -> X20BM11l.SL1]
  InputFilter = 250
PLK1_IOR01SL03 : X20DI6371 v1.1.0.0  [SS1 -> X20TB12c.SS; SL -> X20BM11c.SL1]
  InputFilter = 250
PLK1_IOR01SL04 : X20DI6371 v1.1.0.0  [SS1 -> X20TB12ab.SS; SL -> X20BM11x.SL1]
  InputFilter = 250
PLK1_IOR01SL05 : X20DS1119 v1.4.1.0  [SS1 -> X20TB12e.SS; SL -> X20BM11e.SL1]
  PSInfo = on
  SDCInfo = on
  NetworkInfo = 8Bit
  Function03 = AB
PLK1_IOR01SL07 : X20DO6322 v1.1.0.0  [SS1 -> X20TB12p.SS; SL -> X20cBM11a.SL1]
PLK1_IOR01SL08 : X20DO6322 v1.1.0.0  [SS1 -> X20TB12h.SS; SL -> X20BM11h.SL1]
PLK1_IOR01SL09 : X20ZF0000 v1.1.0.0 (Disabled=true)  [SS1 -> X20TB12o.SS; SL -> X20BM11n.SL1]
PLK1_IOR01SL10 : X20ZF0000 v1.1.0.0 (Disabled=true)  [SS1 -> X20TB12i.SS; SL -> X20BM11m.SL1]
PLK1_IOR01SL11 : X20PS3300 v1.2.0.0  [SS1 -> X20TB12z.SS; SL -> X20BM01.SL1]
  PowerInfo = on
PLK1_IOR01SL12 : X20DI6371 v1.1.0.0  [SS1 -> X20TB12d.SS; SL -> X20BM11d.SL1]
PLK1_IOR01SL13 : X20DO6322 v1.1.0.0  [SS1 -> X20TB12b.SS; SL -> X20BM11b.SL1]
  Supervision = off
PLK1_IOR01SL14 : X20ZF0000 v1.1.0.0 (Disabled=true)  [SS1 -> X20TB12f.SS; SL -> X20BM11f.SL1]
PLK1_IOR01SL15 : X20ZF0000 v1.1.0.0 (Disabled=true)  [SS1 -> X20TB12q.SS; SL -> X20BM11o.SL1]
PLK1_IOR01SL16 : X20SI4100 v2.3.1.0  [SS1 -> X20TB52b.SS; SL -> X20BM33b.SL1]
  SafeModuleID = 116
PLK1_IOR01SL17 : X20SI4100 v2.3.1.0  [SS1 -> X20TB52a.SS; SL -> X20BM33a.SL1]
  SafeModuleID = 117
PLK240-2 : X20IF1082-2 v1.11.1.0  [PLK2 -> BC_PLK1.PLK1 [Cable Type=PowerlinkCable, Length=10, Version=1.0.0.3]; SS -> MCP1_PLC_201.SS1]
  Connector IF1:
    EplHostName = PLC_MCP1_PLK2
    NodeDefinition = Software
    EplNatSubnet = 192.168.102.0
PLK2_IOR02SL02 : X20DI4371 v1.1.0.0  [SS1 -> X20TB12s.SS; SL -> X20BM11p.SL1]
PLK2_IOR02SL03 : X20DI4371 v1.1.0.0  [SS1 -> X20TB12t.SS; SL -> X20BM11q.SL1]
PLK2_IOR02SL04 : X20AI4632-1 v1.1.0.0  [SS1 -> X20TB12u.SS; SL -> X20BM11r.SL1]
  ChannelType01 = 0 to 22mA
  ChannelType02 = 0 to 22mA
  Channel03enable = off
  Channel04enable = off
PLK2_IOR02SL05 : X20DS438A v2.0.1.0  [SS1 -> X20TB12aa.SS; SL -> X20BM11w.SL1]
  DtmRef = FBD.BRIOLinkModuleDTM.DTMCore.X20DS438A
  DtmId = 7db43003-0ff5-4bbd-8923-86eacecae911
  CommDtmId = ab9d1316-8c35-4493-ab34-f7b1b8ca9169
  RequiresDTMBuild = true
  ConfigFile = Communication.dtm
  ConfigModule = asiol1
  OperatingMode01 = Operate
  PDI_Enable01 = variousTypes
  PDI_DataType01_1 = UINT
  OperatingMode02 = Operate
  PDI_Enable02 = variousTypes
  PDI_DataType02_1 = UINT
PLK2_IOR02SL06 : X20PD2113 v1.1.0.0  [SS1 -> X20TB12g.SS; SL -> X20BM11g.SL1]
PLK2_IOR02SL07 : X20ZF0000 v1.1.0.0 (Disabled=true)  [SS1 -> X20TB12x.SS; SL -> X20BM11t.SL1]
PLK2_IOR02SL08 : X20ZF0000 v1.1.0.0 (Disabled=true)  [SS1 -> X20TB12w.SS; SL -> X20BM11v.SL1]
PLK2_IOR02SL09 : X20PS3300 v1.2.0.0 (Disabled=true)  [SS1 -> X20TB12ac.SS; SL -> X20BM01a.SL1]
  PowerInfo = on
PLK2_IOR02SL10 : X20ZF0000 v1.1.0.0 (Disabled=true)  [SS1 -> X20TB12y.SS; SL -> X20BM11u.SL1]
PLK2_IOR02SL11 : X20ZF0000 v1.1.0.0 (Disabled=true)  [SS1 -> X20TB12v.SS; SL -> X20BM11s.SL1]
PLK2_IOR02SL12 : X20SI4100 v2.3.1.0  [SS1 -> X20TB52c.SS; SL -> X20BM33c.SL1]
  SafeModuleID = 212
PLK2_IOR02SL13 : X20SO4120 v2.2.1.0  [SS1 -> X20TB52e.SS; SL -> X20BM33e.SL1]
  PLCopenInfo = on
  SafeModuleID = 213
  DigitalOutput01 = viaSafeLOGIC
  DigitalOutput02 = viaSafeLOGIC
  DigitalOutput03 = viaSafeLOGIC
  DigitalOutput04 = viaSafeLOGIC
PS51x_100_LI2UPN8_IODD1_1 : FBD.IOLink.GenericDeviceDTM.DTMCore.PS51x-100-LI2UPN8 IODD1.1 v2.9 (OrderNumber=PS51x-100-LI2UPN8 IODD1.1)  [IO-Link1 -> PLK2_IOR02SL05.IF1]
  DtmId = 9f03f336-de2c-4174-a814-ce0739b6707c
PS51x_100_LI2UPN8_IODD1_1a : FBD.IOLink.GenericDeviceDTM.DTMCore.PS51x-100-LI2UPN8 IODD1.1 v2.9 (OrderNumber=PS51x-100-LI2UPN8 IODD1.1)  [IO-Link1 -> PLK2_IOR02SL05.IF2]
  DtmId = 948ae1a5-f93f-40dc-8e06-a46fa964d649
PS_PLK1 : X20PS9400 v1.5.0.0  [SS1 -> X20TB12m.SS; PS -> RIO_OWS1_PLK1.PS1]
  PowerInfo = on
PS_PLK2 : X20PS9400 v1.5.0.0  [SS1 -> X20TB12r.SS; PS -> RIO_JB1_PLK2.PS1]
RIO_JB1_PLK2 : X20BB81 v1.0.2.0
RIO_OWS1_PLK1 : X20BB81 v1.0.2.0
SDR1_PLK11 : 8EI2X2HWTS0.xxxx-1 v2.3.1.2  [PLK1 -> MCP1_PLC_201.IF3 (NodeNumber=11) [Cable Type=PowerlinkCable, Length=10, Version=1.0.0.3]; PLK2 -> SDR2_PLK12.PLK1 (NodeNumber=11) [Cable Type=PowerlinkCable, Length=10, Version=1.0.0.3]; EC1 -> ServoMotor_Spindle.EC; EC2 -> ServoMotor_OutE.EC; EC3 -> ServoMotor_InE.EC; MT2 -> ServoMotor_OutE.MT; MT3 -> ServoMotor_InE.MT]
  DriveConfiguration/Module:
    McAcoposTypeID = AcoposP3TConfig
    ActivateACOPOSSimulationOnPLC = 1
  DriveConfiguration/Channel[1]/RealAxis:
    AxisReference = gAxSpin
  DriveConfiguration/Channel[1]/RealAxis/MechanicalElements/Gearbox:
    InputIsReadOnly = 0
    Input = 3
    OutputIsReadOnly = 0
    Output = 1
  DriveConfiguration/Channel[1]/RealAxis/MechanicalElements/RotaryToLinearTransformation:
    ReferenceDistanceIsReadOnly = 0
    ReferenceDistance = 1
  DriveConfiguration/Channel[1]/RealAxis/Controller:
    ModeIsReadOnly = 0
    Mode = PositionController
  DriveConfiguration/Channel[1]/RealAxis/Controller/Mode/Position:
    ProportionalGain = 50.0
    IntegrationTime = 0.0
    PredictionTime = 0.0004
    TotalDelayTime = 0.0004
  DriveConfiguration/Channel[1]/RealAxis/Controller/Mode/Speed:
    ProportionalGainIsReadOnly = 0
    ProportionalGain = 2.0
    IntegrationTimeIsReadOnly = 0
    IntegrationTime = 0.0
    FilterTimeIsReadOnly = 0
    FilterTime = 0.0
  DriveConfiguration/Channel[1]/RealAxis/Controller/Mode/LoopFilters:
    LoopFilter1 = NotUsed
    LoopFilter2 = NotUsed
    LoopFilter3 = NotUsed
  DriveConfiguration/Channel[1]/RealAxis/Homing:
    Mode = Direct
  DriveConfiguration/Channel[1]/RealAxis/Homing/Mode:
    Position = 0.0
    ReferencePulse = NotUsed
  DriveConfiguration/Channel[1]/RealAxis/Homing:
    RestorePositionVariable = 
  DriveConfiguration/Channel[1]/RealAxis/StopReaction:
    Quickstop = DecelerationLimit
    DriveError = DecelerationLimit
  DriveConfiguration/Channel[1]/RealAxis/MovementErrorLimits:
    PositionError = 1.0
    VelocityErrorMonitoring = Automatic1
  DriveConfiguration/Channel[1]/RealAxis:
    JerkFilter = NotUsed
  DriveConfiguration/Channel[1]/RealAxis/DigitalInputs/HomingSwitch:
    Source = NotUsed
    Level = High
  DriveConfiguration/Channel[1]/RealAxis/DigitalInputs/PositiveLimitSwitch:
    Source = NotUsed
    Level = High
  DriveConfiguration/Channel[1]/RealAxis/DigitalInputs/NegativeLimitSwitch:
    Source = NotUsed
    Level = High
  DriveConfiguration/Channel[1]/RealAxis/DigitalInputs/Trigger1:
    Source = NotUsed
    Level = High
  DriveConfiguration/Channel[1]/RealAxis/DigitalInputs/Trigger2:
    Source = NotUsed
    Level = High
  DriveConfiguration/Channel[1]/RealAxis/DigitalInputs/Quickstop:
    Input = NotUsed
  DriveConfiguration/Channel[1]/RealAxis/Simulation:
    SimulationModeOnPLC = SetValueGeneration
    SimulationModeOnACOPOS = NotUsed
  DriveConfiguration/Channel[1]:
    ExternalEncoderAxis = NotUsed
  DriveConfiguration/Channel[2]/RealAxis:
    AxisReference = gAxOutE
  DriveConfiguration/Channel[2]/RealAxis/MechanicalElements/Gearbox:
    InputIsReadOnly = 0
    Input = 5
    OutputIsReadOnly = 0
    Output = 1
  DriveConfiguration/Channel[2]/RealAxis/MechanicalElements/RotaryToLinearTransformation:
    ReferenceDistanceIsReadOnly = 0
    ReferenceDistance = 360.0
  DriveConfiguration/Channel[2]/RealAxis/Controller:
    ModeIsReadOnly = 0
    Mode = PositionController
  DriveConfiguration/Channel[2]/RealAxis/Controller/Mode/Position:
    ProportionalGain = 50.0
    IntegrationTime = 0.0
    PredictionTime = 0.0004
    TotalDelayTime = 0.0004
  DriveConfiguration/Channel[2]/RealAxis/Controller/Mode/Speed:
    ProportionalGainIsReadOnly = 0
    ProportionalGain = 2.0
    IntegrationTimeIsReadOnly = 0
    IntegrationTime = 0.0
    FilterTimeIsReadOnly = 0
    FilterTime = 0.0
  DriveConfiguration/Channel[2]/RealAxis/Controller/Mode/LoopFilters:
    LoopFilter1 = NotUsed
    LoopFilter2 = NotUsed
    LoopFilter3 = NotUsed
  DriveConfiguration/Channel[2]/RealAxis/Homing:
    Mode = Direct
  DriveConfiguration/Channel[2]/RealAxis/Homing/Mode:
    Position = 0.0
    ReferencePulse = NotUsed
  DriveConfiguration/Channel[2]/RealAxis/Homing:
    RestorePositionVariable = ::gr_AxOutERestorePos
  DriveConfiguration/Channel[2]/RealAxis/StopReaction:
    Quickstop = DecelerationLimit
    DriveError = DecelerationLimit
  DriveConfiguration/Channel[2]/RealAxis/MovementErrorLimits:
    PositionError = 1.0
    VelocityErrorMonitoring = Automatic1
  DriveConfiguration/Channel[2]/RealAxis:
    JerkFilter = NotUsed
  DriveConfiguration/Channel[2]/RealAxis/DigitalInputs/HomingSwitch:
    Source = NotUsed
    Level = High
  DriveConfiguration/Channel[2]/RealAxis/DigitalInputs/PositiveLimitSwitch:
    Source = NotUsed
    Level = High
  DriveConfiguration/Channel[2]/RealAxis/DigitalInputs/NegativeLimitSwitch:
    Source = NotUsed
    Level = High
  DriveConfiguration/Channel[2]/RealAxis/DigitalInputs/Trigger1:
    Source = NotUsed
    Level = High
  DriveConfiguration/Channel[2]/RealAxis/DigitalInputs/Trigger2:
    Source = NotUsed
    Level = High
  DriveConfiguration/Channel[2]/RealAxis/DigitalInputs/Quickstop:
    Input = Trigger2
  DriveConfiguration/Channel[2]/RealAxis/Simulation:
    SimulationModeOnPLC = SetValueGeneration
    SimulationModeOnACOPOS = NotUsed
  DriveConfiguration/Channel[2]:
    ExternalEncoderAxis = NotUsed
  DriveConfiguration/Channel[3]/RealAxis:
    AxisReference = gAxInE
  DriveConfiguration/Channel[3]/RealAxis/MechanicalElements/Gearbox:
    InputIsReadOnly = 0
    Input = 5
    OutputIsReadOnly = 0
    Output = 1
  DriveConfiguration/Channel[3]/RealAxis/MechanicalElements/RotaryToLinearTransformation:
    ReferenceDistanceIsReadOnly = 0
    ReferenceDistance = 360.0
  DriveConfiguration/Channel[3]/RealAxis/Controller:
    ModeIsReadOnly = 0
    Mode = PositionController
  DriveConfiguration/Channel[3]/RealAxis/Controller/Mode/Position:
    ProportionalGain = 50.0
    IntegrationTime = 0.0
    PredictionTime = 0.0004
    TotalDelayTime = 0.0004
  DriveConfiguration/Channel[3]/RealAxis/Controller/Mode/Speed:
    ProportionalGainIsReadOnly = 0
    ProportionalGain = 2.0
    IntegrationTimeIsReadOnly = 0
    IntegrationTime = 0.0
    FilterTimeIsReadOnly = 0
    FilterTime = 0.0
  DriveConfiguration/Channel[3]/RealAxis/Controller/Mode/LoopFilters:
    LoopFilter1 = NotUsed
    LoopFilter2 = NotUsed
    LoopFilter3 = NotUsed
  DriveConfiguration/Channel[3]/RealAxis/Homing:
    Mode = Direct
  DriveConfiguration/Channel[3]/RealAxis/Homing/Mode:
    Position = 0.0
    ReferencePulse = NotUsed
  DriveConfiguration/Channel[3]/RealAxis/Homing:
    RestorePositionVariable = ::gr_AxInERestorePos
  DriveConfiguration/Channel[3]/RealAxis/StopReaction:
    Quickstop = DecelerationLimit
    DriveError = DecelerationLimit
  DriveConfiguration/Channel[3]/RealAxis/MovementErrorLimits:
    PositionError = 1.0
    VelocityErrorMonitoring = Automatic1
  DriveConfiguration/Channel[3]/RealAxis:
    JerkFilter = NotUsed
  DriveConfiguration/Channel[3]/RealAxis/DigitalInputs/HomingSwitch:
    Source = NotUsed
    Level = High
  DriveConfiguration/Channel[3]/RealAxis/DigitalInputs/PositiveLimitSwitch:
    Source = NotUsed
    Level = High
  DriveConfiguration/Channel[3]/RealAxis/DigitalInputs/NegativeLimitSwitch:
    Source = NotUsed
    Level = High
  DriveConfiguration/Channel[3]/RealAxis/DigitalInputs/Trigger1:
    Source = NotUsed
    Level = High
  DriveConfiguration/Channel[3]/RealAxis/DigitalInputs/Trigger2:
    Source = NotUsed
    Level = High
  DriveConfiguration/Channel[3]/RealAxis/DigitalInputs/Quickstop:
    Input = NotUsed
  DriveConfiguration/Channel[3]/RealAxis/Simulation:
    SimulationModeOnPLC = SetValueGeneration
    SimulationModeOnACOPOS = NotUsed
  DriveConfiguration/Channel[3]:
    ExternalEncoderAxis = NotUsed
SDR2_PLK12 : 8EI8X8HWSS0.xxxx-1 v2.3.1.2  [PLK1 -> SDR1_PLK11.PLK2 (NodeNumber=12) [Cable Type=PowerlinkCable, Length=10, Version=1.0.0.3]; PLK2 -> VFD1_PLK13.PLK1 (NodeNumber=12) [Cable Type=PowerlinkCable, Length=10, Version=1.0.0.3]; EC1 -> ServoMotor_Z.EC]
  DriveConfiguration/Module:
    McAcoposTypeID = AcoposP3SConfig
    ActivateACOPOSSimulationOnPLC = 1
  DriveConfiguration/Channel[1]/RealAxis:
    AxisReference = gAxZ
  DriveConfiguration/Channel[1]/RealAxis/MechanicalElements/Gearbox:
    InputIsReadOnly = 0
    Input = 1
    OutputIsReadOnly = 0
    Output = 1
  DriveConfiguration/Channel[1]/RealAxis/MechanicalElements/RotaryToLinearTransformation:
    ReferenceDistanceIsReadOnly = 0
    ReferenceDistance = 2.54
  DriveConfiguration/Channel[1]/RealAxis/Controller:
    ModeIsReadOnly = 0
    Mode = PositionController
  DriveConfiguration/Channel[1]/RealAxis/Controller/Mode/Position:
    ProportionalGain = 50.0
    IntegrationTime = 0.0
    PredictionTime = 0.0004
    TotalDelayTime = 0.0004
  DriveConfiguration/Channel[1]/RealAxis/Controller/Mode/Speed:
    ProportionalGainIsReadOnly = 0
    ProportionalGain = 2.0
    IntegrationTimeIsReadOnly = 0
    IntegrationTime = 0.0
    FilterTimeIsReadOnly = 0
    FilterTime = 0.0
  DriveConfiguration/Channel[1]/RealAxis/Controller/Mode/LoopFilters:
    LoopFilter1 = NotUsed
    LoopFilter2 = NotUsed
    LoopFilter3 = NotUsed
  DriveConfiguration/Channel[1]/RealAxis/Homing:
    Mode = Direct
  DriveConfiguration/Channel[1]/RealAxis/Homing/Mode:
    Position = 0.0
    ReferencePulse = NotUsed
  DriveConfiguration/Channel[1]/RealAxis/Homing:
    RestorePositionVariable = ::gr_AxZRestorePos
  DriveConfiguration/Channel[1]/RealAxis/StopReaction:
    Quickstop = DecelerationLimit
    DriveError = DecelerationLimit
  DriveConfiguration/Channel[1]/RealAxis/MovementErrorLimits:
    PositionError = 1.0
    VelocityErrorMonitoring = Automatic1
  DriveConfiguration/Channel[1]/RealAxis:
    JerkFilter = NotUsed
  DriveConfiguration/Channel[1]/RealAxis/DigitalInputs/HomingSwitch:
    Source = NotUsed
    Level = High
  DriveConfiguration/Channel[1]/RealAxis/DigitalInputs/PositiveLimitSwitch:
    Source = X8Trigger1
    Level = High
  DriveConfiguration/Channel[1]/RealAxis/DigitalInputs/NegativeLimitSwitch:
    Source = X8Trigger2
    Level = High
  DriveConfiguration/Channel[1]/RealAxis/DigitalInputs/Trigger1:
    Source = NotUsed
    Level = High
  DriveConfiguration/Channel[1]/RealAxis/DigitalInputs/Trigger2:
    Source = NotUsed
    Level = High
  DriveConfiguration/Channel[1]/RealAxis/DigitalInputs/Quickstop:
    Input = NotUsed
  DriveConfiguration/Channel[1]/RealAxis/Simulation:
    SimulationModeOnPLC = SetValueGeneration
    SimulationModeOnACOPOS = NotUsed
  DriveConfiguration/Channel[1]:
    ExternalEncoderAxis = NotUsed
SafetyController_R01SL06 : X20SLX410 v2.4.0.1  [SS1 -> X20TB52.SS; SL -> X20BM33.SL1]
  UnsafeOutputBOOLs = 16
  UnsafeInputBOOLs = 24
  UnsafeInputUINTs = 4
ServoMotor_InE : 8LSA26.D9060S200-3 v2.2.0.1  [EC -> SDR1_PLK11.EC3; MT -> SDR1_PLK11.MT3]
  M1/MotorParameters:
    MOTOR_AMB_TEMP_RATED = 40
ServoMotor_OutE : 8LSA26.D9060S200-3 v2.2.0.1  [EC -> SDR1_PLK11.EC2; MT -> SDR1_PLK11.MT2]
  M1/MotorParameters:
    MOTOR_AMB_TEMP_RATED = 40
ServoMotor_Spindle : 8LSA26.D9060S200-3 v2.2.0.1  [EC -> SDR1_PLK11.EC1; MT -> SDR1_PLK11.MT1]
  M1/MotorParameters:
    MOTOR_AMB_TEMP_RATED = 40
ServoMotor_Z : 8LSA46.DB030S200-3 v1.0.8.37  [EC -> SDR2_PLK12.EC1; MT -> SDR2_PLK12.MT1]
  M1/MotorParameters:
    MOTOR_AMB_TEMP_RATED = 40
VFD1_PLK13 : 8I66xxxxxxx.0P-xxx v2.3.2.0  [PLK1 -> SDR2_PLK12.PLK2 [Cable Type=PowerlinkCable, Length=10, Version=1.0.0.3]]
  FunctionModel = MotionConfig
  Supervision = off
  McTypeID = McAcoposInverterP66P
  AxisReference = gAxCfPmp
  InputIsReadOnly = 0
  Input = 1
  OutputIsReadOnly = 0
  Output = 1
  ReferenceDistanceIsReadOnly = 0
  ReferenceDistance = 1
  UnitOfSetpoint = Rpm
  Mode_LI3 = Safety
  Sel_NameplateMask = 8Ix6T401100_IEC
  Cfg_NSP = 1175
  Cfg_FRS = 600
  Cfg_UNS = 480
  Cfg_COS = 73
X20BM01 : X20BM01 v2.1.0.0  [X2X1 -> X20BM11m.X2X2]
X20BM01a : X20BM01 v2.1.0.0 (Disabled=true)  [X2X1 -> X20BM11v.X2X2]
X20BM11 : X20BM11 v1.1.0.0  [X2X1 -> MCP1_PLC_201.IF6]
X20BM11b : X20BM11 v1.1.0.0  [X2X1 -> X20BM11d.X2X2]
X20BM11c : X20BM11 v1.1.0.0  [X2X1 -> X20BM11l.X2X2]
X20BM11d : X20BM11 v1.1.0.0  [X2X1 -> X20BM01.X2X2]
X20BM11e : X20BM11 v1.1.0.0  [X2X1 -> X20BM11x.X2X2]
X20BM11f : X20BM11 v1.1.0.0 (Disabled=true)  [X2X1 -> X20BM11b.X2X2]
X20BM11g : X20BM11 v1.1.0.0  [X2X1 -> X20BM11w.X2X2]
X20BM11h : X20BM11 v1.1.0.0  [X2X1 -> X20cBM11a.X2X2]
X20BM11l : X20BM11 v1.1.0.0  [X2X1 -> RIO_OWS1_PLK1.IF1]
X20BM11m : X20BM11 v1.1.0.0 (Disabled=true)  [X2X1 -> X20BM11n.X2X2]
X20BM11n : X20BM11 v1.1.0.0 (Disabled=true)  [X2X1 -> X20BM11h.X2X2]
X20BM11o : X20BM11 v1.1.0.0 (Disabled=true)  [X2X1 -> X20BM11f.X2X2]
X20BM11p : X20BM11 v1.1.0.0  [X2X1 -> RIO_JB1_PLK2.IF1]
X20BM11q : X20BM11 v1.1.0.0  [X2X1 -> X20BM11p.X2X2]
X20BM11r : X20BM11 v1.1.0.0  [X2X1 -> X20BM11q.X2X2]
X20BM11s : X20BM11 v1.1.0.0 (Disabled=true)  [X2X1 -> X20BM11u.X2X2]
X20BM11t : X20BM11 v1.1.0.0 (Disabled=true)  [X2X1 -> X20BM11g.X2X2]
X20BM11u : X20BM11 v1.1.0.0 (Disabled=true)  [X2X1 -> X20BM01a.X2X2]
X20BM11v : X20BM11 v1.1.0.0 (Disabled=true)  [X2X1 -> X20BM11t.X2X2]
X20BM11w : X20BM11 v1.1.0.0  [X2X1 -> X20BM11r.X2X2]
X20BM11x : X20BM11 v1.1.0.0  [X2X1 -> X20BM11c.X2X2]
X20BM33 : X20BM33 v1.0.0.6  [X2X1 -> X20BM11e.X2X2]
X20BM33a : X20BM33 v1.0.0.6  [X2X1 -> X20BM33b.X2X2]
X20BM33b : X20BM33 v1.0.0.6  [X2X1 -> X20BM11o.X2X2]
X20BM33c : X20BM33 v1.0.0.6  [X2X1 -> X20BM11s.X2X2]
X20BM33d : X20BM33 v1.0.0.6  [X2X1 -> X20BM11.X2X2]
X20BM33e : X20BM33 v1.0.0.6  [X2X1 -> X20BM33c.X2X2]
X20TB12 : X20TB12 v1.0.0.0
X20TB12aa : X20TB12 v1.0.0.0
X20TB12ab : X20TB12 v1.0.0.0
X20TB12ac : X20TB12 v1.0.0.0 (Disabled=true)
X20TB12b : X20TB12 v1.0.0.0
X20TB12c : X20TB12 v1.0.0.0
X20TB12d : X20TB12 v1.0.0.0
X20TB12e : X20TB12 v1.0.0.0
X20TB12f : X20TB12 v1.0.0.0 (Disabled=true)
X20TB12g : X20TB12 v1.0.0.0
X20TB12h : X20TB12 v1.0.0.0
X20TB12i : X20TB12 v1.0.0.0 (Disabled=true)
X20TB12m : X20TB12 v1.0.0.0
X20TB12n : X20TB12 v1.0.0.0
X20TB12o : X20TB12 v1.0.0.0 (Disabled=true)
X20TB12p : X20TB12 v1.0.0.0
X20TB12q : X20TB12 v1.0.0.0 (Disabled=true)
X20TB12r : X20TB12 v1.0.0.0
X20TB12s : X20TB12 v1.0.0.0
X20TB12t : X20TB12 v1.0.0.0
X20TB12u : X20TB12 v1.0.0.0
X20TB12v : X20TB12 v1.0.0.0 (Disabled=true)
X20TB12w : X20TB12 v1.0.0.0 (Disabled=true)
X20TB12x : X20TB12 v1.0.0.0 (Disabled=true)
X20TB12y : X20TB12 v1.0.0.0 (Disabled=true)
X20TB12z : X20TB12 v1.0.0.0
X20TB52 : X20TB52 v1.0.0.2
X20TB52a : X20TB52 v1.0.0.2
X20TB52b : X20TB52 v1.0.0.2
X20TB52c : X20TB52 v1.0.0.2
X20TB52d : X20TB52 v1.0.0.2
X20TB52e : X20TB52 v1.0.0.2
X20cBM11a : X20cBM11 v1.0.1.0  [X2X1 -> X20BM33.X2X2]
```

### Cpu.per - MCP1_PLC_201/Cpu.per
```iecst
VAR_CONFIG
	gr_AxOutERestorePos AT %M0; (* *)
	gr_AxInERestorePos AT %M72; (* *)
	gr_AxZRestorePos AT %M144; (* *)
	gr_AI_FT_CFFlow_Params AT %M216; (* *)
	gr_AI_LT_CFTankLevel_Params AT %M304; (* *)
	gr_AI_PT_CFFilterOutlet_Params AT %M392; (* *)
	gr_AI_PT_CFPumpOutlet_Params AT %M480; (* *)
	gr_AI_DP_CFFilter_Params AT %M568; (* *)
	gr_DI_JI_480VACOk_Params AT %M656; (* *)
	gr_DI_LSL_CFTank_Params AT %M688; (* *)
	gr_DI_ZS_CFTankLocator_Params AT %M720; (* *)
	gr_AxisPositionLimits AT %M752; (* *)
	gr_CfgCurrent AT %M896; (* *)
	gr_PartCurrent AT %M1080; (* *)
END_VAR
```

### Simple.dob - MCP1_PLC_201/DataObject/Simple.dob
```
DataObject (SubType=Simple)
  Files:
    File = DataObject.dat
```

### IoMap.iom - MCP1_PLC_201/IoMap.iom
```iecst
VAR_CONFIG
	::AI_FT_CFFlow.InRawINT AT %IW."PLK2_IOR02SL04".AnalogInput01;
	::AI_FT_CFFlow.ChannelOk AT %IX."PLK2_IOR02SL04".Channel01OK INVERSE;
	::AI_LT_CFTankLevel.InRawINT AT %IW."PLK2_IOR02SL04".AnalogInput02;
	::AI_LT_CFTankLevel.ChannelOk AT %IX."PLK2_IOR02SL04".Channel02OK INVERSE;
	::ModStat_JB1_PLK2.Slot05ModuleOk AT %IX."PLK2_IOR02SL05".ModuleOk;
	::ModStat_JB1_PLK2.Slot02ModuleOk AT %IX."PLK2_IOR02SL02".ModuleOk;
	::ModStat_JB1_PLK2.Slot03ModuleOk AT %IX."PLK2_IOR02SL03".ModuleOk;
	::ModStat_JB1_PLK2.Slot04ModuleOk AT %IX."PLK2_IOR02SL04".ModuleOk;
	::ModStat_JB1_PLK2.Slot06ModuleOk AT %IX."PLK2_IOR02SL06".ModuleOk;
	::ModStat_JB1_PLK2.Slot09ModuleOk AT %IX."PLK2_IOR02SL09".ModuleOk;
	::ModStat_JB1_PLK2.Slot12ModuleOk AT %IX."PLK2_IOR02SL12".ModuleOk;
	::ModStat_JB1_PLK2.Slot13ModuleOk AT %IX."PLK2_IOR02SL13".ModuleOk;
	::ModStat_OWS_PLK1.Slot02ModuleOk AT %IX."PLK1_IOR01SL02".ModuleOk;
	::ModStat_OWS_PLK1.Slot03ModuleOk AT %IX."PLK1_IOR01SL03".ModuleOk;
	::ModStat_OWS_PLK1.Slot04ModuleOk AT %IX."PLK1_IOR01SL04".ModuleOk;
	::ModStat_OWS_PLK1.Slot05ModuleOk AT %IX."PLK1_IOR01SL05".ModuleOk;
	::ModStat_OWS_PLK1.Slot07ModuleOk AT %IX."PLK1_IOR01SL07".ModuleOk;
	::ModStat_OWS_PLK1.Slot08ModuleOk AT %IX."PLK1_IOR01SL08".ModuleOk;
	::ModStat_OWS_PLK1.Slot11ModuleOk AT %IX."PLK1_IOR01SL11".ModuleOk;
	::ModStat_OWS_PLK1.Slot12ModuleOk AT %IX."PLK1_IOR01SL12".ModuleOk;
	::ModStat_OWS_PLK1.Slot13ModuleOk AT %IX."PLK1_IOR01SL13".ModuleOk;
	::ModStat_OWS_PLK1.Slot16ModuleOk AT %IX."PLK1_IOR01SL16".ModuleOk;
	::ModStat_OWS_PLK1.Slot17ModuleOk AT %IX."PLK1_IOR01SL17".ModuleOk;
	::ModStat_PLC_201.Slot01ModuleOk AT %IX."IOR00SL01".ModuleOk;
	::ModStat_OWS_PLK1.Slot06ModuleOk AT %IX."SafetyController_R01SL06".ModuleOk;
	::DI_LSL_CFTank.InRaw AT %IX."PLK2_IOR02SL02".DigitalInput01;
	::DI_ZS_CFTankLocator.InRaw AT %IX."PLK2_IOR02SL02".DigitalInput02;
	::DI_JI_480VACOk.InRaw AT %IX."IOR00SL01".DigitalInput01;
	::owsPendant.AxisSelectInputs[1] AT %IX."PLK1_IOR01SL02".DigitalInput01;
	::owsPendant.AxisSelectInputs[2] AT %IX."PLK1_IOR01SL02".DigitalInput02;
	::owsPendant.AxisSelectInputs[3] AT %IX."PLK1_IOR01SL02".DigitalInput03;
	::owsPendant.SpeedSelectInputs[1] AT %IX."PLK1_IOR01SL02".DigitalInput04;
	::owsPendant.SpeedSelectInputs[2] AT %IX."PLK1_IOR01SL02".DigitalInput05;
	::owsPendant.SpeedSelectInputs[3] AT %IX."PLK1_IOR01SL02".DigitalInput06;
	::owsPendant.PBInputs[1] AT %IX."PLK1_IOR01SL03".DigitalInput01;
	::owsPendant.PBInputs[2] AT %IX."PLK1_IOR01SL03".DigitalInput02;
	::owsPendant.PBInputs[3] AT %IX."PLK1_IOR01SL03".DigitalInput03;
	::owsPendant.PBInputs[4] AT %IX."PLK1_IOR01SL03".DigitalInput04;
	::owsPendant.PBInputs[5] AT %IX."PLK1_IOR01SL03".DigitalInput05;
	::owsPendant.PBInputs[6] AT %IX."PLK1_IOR01SL03".DigitalInput06;
	::owsPendant.PBInputs[7] AT %IX."PLK1_IOR01SL04".DigitalInput01;
	::owsPendant.PBInputs[8] AT %IX."PLK1_IOR01SL04".DigitalInput02;
	::owsPendant.PBInputs[9] AT %IX."PLK1_IOR01SL04".DigitalInput03;
	::owsPendant.tmrCountResetPulse.Q AT %QX."PLK1_IOR01SL05".CounterReset;
	::owsPendant.encoderPowerOk AT %IX."PLK1_IOR01SL05".PowerSupply02 INVERSE;
	::owsPendant.HandwheelCounter AT %ID."PLK1_IOR01SL05".CounterValue01;
	::axes[1].Status.SafeMotionDiagCode AT %IW."SafetyController_R01SL06".UINT0001;
	::axes[2].Status.SafeMotionDiagCode AT %IW."SafetyController_R01SL06".UINT0002;
	::axes[3].Status.SafeMotionDiagCode AT %IW."SafetyController_R01SL06".UINT0003;
	::axes[4].Status.SafeMotionDiagCode AT %IW."SafetyController_R01SL06".UINT0004;
	::OmSafeDev:fs_EmoCmd AT %IX."SafetyController_R01SL06".BOOL00001;
	::OmSafeDev:fs_AllSMsOk AT %IX."SafetyController_R01SL06".BOOL00002;
	::OmSafeDev:fs_EmoOwsOk AT %IX."SafetyController_R01SL06".BOOL00007;
	::owsPendant.emoAcivated AT %IX."SafetyController_R01SL06".BOOL00008;
	::OmSafeDev:fs_StartPbOk AT %IX."SafetyController_R01SL06".BOOL00013;
	::OmSafeDev:fs_KeyswitchInRun AT %IX."SafetyController_R01SL06".BOOL00014;
	::OmSafeDev:fs_KeyswitchOk AT %IX."SafetyController_R01SL06".BOOL00015;
	::owsPendant.enableSwActive AT %IX."SafetyController_R01SL06".BOOL00017;
	::OmSafeDev:fs_CfGateClosed AT %IX."SafetyController_R01SL06".BOOL00019;
	::axes[4].Commands.ReleaseBrakeCmd AT %QX."SafetyController_R01SL06".BOOL10016;
	::axes[3].Commands.ReleaseBrakeCmd AT %QX."SafetyController_R01SL06".BOOL10015;
	::axes[2].Commands.ReleaseBrakeCmd AT %QX."SafetyController_R01SL06".BOOL10014;
	::axes[1].Commands.ReleaseBrakeCmd AT %QX."SafetyController_R01SL06".BOOL10013;
	::OmSafeDev:ts_ResetEStop AT %QX."SafetyController_R01SL06".BOOL10001;
	::OmSafeDev:ts_ResetSafeMC AT %QX."SafetyController_R01SL06".BOOL10002;
	::axes[1].Commands.PlcSafetyEnable AT %QX."SafetyController_R01SL06".BOOL10008;
	::axes[2].Commands.PlcSafetyEnable AT %QX."SafetyController_R01SL06".BOOL10009;
	::axes[3].Commands.PlcSafetyEnable AT %QX."SafetyController_R01SL06".BOOL10010;
	::axes[4].Commands.PlcSafetyEnable AT %QX."SafetyController_R01SL06".BOOL10011;
	::OmSafeDev:ts_InEmoMode AT %QX."SafetyController_R01SL06".BOOL10003;
	::OmSafeDev:ts_InSafeMode AT %QX."SafetyController_R01SL06".BOOL10004;
	::OmSafeDev:ts_InPendantMode AT %QX."SafetyController_R01SL06".BOOL10005;
	::OmSafeDev:fs_CfGateClosedLocked AT %IX."SafetyController_R01SL06".BOOL00020;
	::DO_PL_OWSGreen AT %QX."PLK1_IOR01SL13".DigitalOutput01;
	::DO_PL_OWSAmber AT %QX."PLK1_IOR01SL13".DigitalOutput02;
	::DO_PL_OWSRed AT %QX."PLK1_IOR01SL13".DigitalOutput03;
	::DO_PL_OWSBeconGreen AT %QX."PLK1_IOR01SL13".DigitalOutput04;
	::DO_PL_OWSBeconAmber AT %QX."PLK1_IOR01SL13".DigitalOutput05;
	::DO_PL_OWSBeconRed AT %QX."PLK1_IOR01SL13".DigitalOutput06;
	::AI_PT_CFPumpOutlet.InRawUINT AT %IW."PLK2_IOR02SL05".InputData01_1;
	::AI_PT_CFFilterOutlet.InRawUINT AT %IW."PLK2_IOR02SL05".InputData02_1;
	::owsPendant.emoWiringOk AT %IX."SafetyController_R01SL06".BOOL00009;
	::OmSafeDev:fs_StopPbActive AT %IX."SafetyController_R01SL06".BOOL00010;
	::owsPendant.pendantAllowMoves AT %IX."SafetyController_R01SL06".BOOL00003;
	::OmSafeDev:fs_EmoOwsActive AT %IX."SafetyController_R01SL06".BOOL00006;
	::OmSafeDev:fs_StopPbOk AT %IX."SafetyController_R01SL06".BOOL00011;
	::OmSafeDev:fs_StartPbActive AT %IX."SafetyController_R01SL06".BOOL00012;
	::owsPendant.enableSwWiringOk AT %IX."SafetyController_R01SL06".BOOL00018;
	::ProdCycle:ts_InCycle AT %QX."SafetyController_R01SL06".BOOL10006;
	::ProdCycle:ts_cfLockGate AT %QX."SafetyController_R01SL06".BOOL10007;
	::OmSafeDev:fs_InSafeMode AT %IX."SafetyController_R01SL06".BOOL00016;
	::ModStat_PLC_201.Slot02ModuleOk AT %IX."IOR00SL02".ModuleOk;
	::owsPendant.PLCmds[1] AT %QX."PLK1_IOR01SL07".DigitalOutput01;
	::owsPendant.PLCmds[2] AT %QX."PLK1_IOR01SL07".DigitalOutput02;
	::owsPendant.PLCmds[3] AT %QX."PLK1_IOR01SL07".DigitalOutput03;
	::owsPendant.PLCmds[4] AT %QX."PLK1_IOR01SL07".DigitalOutput04;
	::owsPendant.PLCmds[5] AT %QX."PLK1_IOR01SL07".DigitalOutput05;
	::owsPendant.PLCmds[6] AT %QX."PLK1_IOR01SL07".DigitalOutput06;
	::owsPendant.PLCmds[7] AT %QX."PLK1_IOR01SL08".DigitalOutput01;
	::owsPendant.PLCmds[8] AT %QX."PLK1_IOR01SL08".DigitalOutput02;
	::owsPendant.PLCmds[9] AT %QX."PLK1_IOR01SL08".DigitalOutput03;
	::DO_PB_OWSGreen AT %QX."PLK1_IOR01SL08".DigitalOutput04;
	::DO_PB_OWSRed AT %QX."PLK1_IOR01SL08".DigitalOutput05;
	::OmSafeDev:fs_CfGateClosedOk AT %IX."SafetyController_R01SL06".BOOL00021;
	::owsPendant.pendantPowerOk AT %IX."PLK1_IOR01SL05".PowerSupply01 INVERSE;
END_VAR
```

### vAxHw.axis - MCP1_PLC_201/mappMotion/Handwheel/vAxHw.axis
```
Element gvAxHw (Type=axis)
  BaseTypeIsReadOnly = 0
  BaseType = RotaryPeriodic
    MeasurementUnitIsReadOnly = 0
    MeasurementUnit = 17476
    MeasurementResolutionIsReadOnly = 0
    MeasurementResolution = 0.01
    CountDirectionIsReadOnly = 0
    CountDirection = Standard
    PeriodSettings:
      Period = 360.0
  MovementLimitsIsReadOnly = 0
  MovementLimits = Internal
    Position:
      LowerLimitMin = -1.79769313486231E308
      UpperLimitMax = 1.79769313486231E308
      LowerLimit = -1000.0
      UpperLimit = 1000.0
    VelocityIsReadOnly = 0
    Velocity:
      VelocityMax = 3.4E38
      Velocity = 10.0
    AccelerationIsReadOnly = 0
    Acceleration:
      AccelerationMax = 3.4E38
      Acceleration = 50.0
    DecelerationIsReadOnly = 0
    Deceleration:
      DecelerationMax = 3.4E38
      Deceleration = 50.0
  Alarms = MpAlarmX
```

### axCfgCfPmp.axis - MCP1_PLC_201/mappMotion/axCfgCfPmp.axis
```
Element gAxCfPmp (Type=axis)
  BaseTypeIsReadOnly = 0
  BaseType = Rotary
    MeasurementUnitIsReadOnly = 0
    MeasurementUnit = 5059636
    MeasurementResolutionIsReadOnly = 0
    MeasurementResolution = 1.0
    CountDirectionIsReadOnly = 0
    CountDirection = Standard
  MovementLimitsIsReadOnly = 0
  MovementLimits = Internal
    Position:
      LowerLimitMin = -1.79769313486231E308
      UpperLimitMax = 1.79769313486231E308
      LowerLimit = -1000.0
      UpperLimit = 1000.0
    VelocityIsReadOnly = 0
    Velocity:
      VelocityMax = 3.4E38
      Velocity = 19.583
    AccelerationIsReadOnly = 0
    Acceleration:
      AccelerationMax = 3.4E38
      Acceleration = 10
    DecelerationIsReadOnly = 0
    Deceleration:
      DecelerationMax = 3.4E38
      Deceleration = 10
  Alarms = MpAlarmX
```

### axCfgOutE.axis - MCP1_PLC_201/mappMotion/axCfgOutE.axis
```
Element gAxOutE (Type=axis)
  BaseTypeIsReadOnly = 0
  BaseType = RotaryPeriodic
    MeasurementUnitIsReadOnly = 0
    MeasurementUnit = 17476
    MeasurementResolutionIsReadOnly = 0
    MeasurementResolution = 0.001
    CountDirectionIsReadOnly = 0
    CountDirection = Standard
    PeriodSettings:
      Period = 360.0
  MovementLimitsIsReadOnly = 0
  MovementLimits = Internal
    Position:
      LowerLimitMin = -1.79769313486231E308
      UpperLimitMax = 1.79769313486231E308
      LowerLimit = -1000.0
      UpperLimit = 1000.0
    VelocityIsReadOnly = 0
    Velocity:
      VelocityMax = 3.4E38
      Velocity = 18
    AccelerationIsReadOnly = 0
    Acceleration:
      AccelerationMax = 3.4E38
      Acceleration = 20
    DecelerationIsReadOnly = 0
    Deceleration:
      DecelerationMax = 3.4E38
      Deceleration = 75
  Alarms = MpAlarmX
```

### axCfgSpin.axis - MCP1_PLC_201/mappMotion/axCfgSpin.axis
```
Element gAxSpin (Type=axis)
  BaseTypeIsReadOnly = 0
  BaseType = RotaryPeriodic
    MeasurementUnitIsReadOnly = 0
    MeasurementUnit = 5059636
    MeasurementResolutionIsReadOnly = 0
    MeasurementResolution = 0.01
    CountDirectionIsReadOnly = 0
    CountDirection = Standard
    PeriodSettings:
      Period = 1.0
  MovementLimitsIsReadOnly = 0
  MovementLimits = Internal
    Position:
      LowerLimitMin = -1.79769313486231E308
      UpperLimitMax = 1.79769313486231E308
      LowerLimit = -1000.0
      UpperLimit = 1000.0
    VelocityIsReadOnly = 0
    Velocity:
      VelocityMax = 3.4E38
      Velocity = 40
    AccelerationIsReadOnly = 0
    Acceleration:
      AccelerationMax = 3.4E38
      Acceleration = 20
    DecelerationIsReadOnly = 0
    Deceleration:
      DecelerationMax = 3.4E38
      Deceleration = 140
  Alarms = MpAlarmX
```

## Logical view

Binary libraries used (declarations not repeated): operator, runtime, standard, brsystem, sys_lib, AsBrMath, AsBrStr, astime, AsIecCon, GAConvert, AsZip, FileIO, McBase, MpAxis, McAcpAx, McPureVAx 5.17.1, McAxis, McDS402Ax 5.17.1, MpBase, SfDomain 5.17.0, MpRecipe, MpAlarmX, CoTrace, MTLookUp 5.17.0

### Global.typ
```iecst
(********************************************************************
 * COPYRIGHT -- General Atomics
 ********************************************************************
 * File: Global.typ
 * Author: J. Sheeron
 ********************************************************************
 * Global data types of project 305841-E00002
 ********************************************************************)

TYPE
  (****************************************)
  (***** Depth to Angle Lookup ************)
  (****************************************)

	sXYTableReal50 : STRUCT
    numberOfVals : USINT := 0; (* number of values defined *)
		xVals : ARRAY[0..49]OF REAL;
		yVals : ARRAY[0..49]OF REAL;
	END_STRUCT;

	sDepthToAngleLu : STRUCT
    T1 : sXYTableReal50;
    T2 : sXYTableReal50;
    T3 : sXYTableReal50;
	END_STRUCT;

  (****************************************)
  (***** Workpiece related structures *****)
  (****************************************)

  (***** Information about a specific part *)

  sWp_Part : STRUCT (* a specific part *)
    isZCalibrated : BOOL; (* position is calibrated to process *)
    isZIndexed : BOOL; (* set when Z is at a proper index -- position is an integer multiple of index distance *)
    isOutECalibrated : BOOL; (* position is calibrated to process *)
    isInECalibrated : BOOL; (* position is calibrated to process *)
    cutPassCount : USINT; (* which cut pass is the process on *)
    zIndexCount : USINT; (* which index is Z on -- An integer rounded version of zIndexLRCount. *)
    zIndexCountSuccess : USINT; (* last index with a successful cut *)
    zIndexLRCount : LREAL; (* which index is Z on -- should normally be an integer. An LREAL for position compatability and so a proper index can be calculated *)
    serialNumber : STRING[25]; (* Part Serial Number *)
    partDfn : sWp_PartDfn; (* Part Definition used for this part *)
  END_STRUCT;

  (***** Information about a configuration or machine setup *)
  sWp_CuttingHead :	STRUCT
    (* changes to cut profile values are detected to enable/disable cam table loading *)
    StartOfCutProfile : BOOL := FALSE;
    finishingPass : BOOL; (* finishing pass yes or no *)
    passCount : USINT; (* number of passes *)
    totalDepth : REAL; (* mm, finished depth *)
    finishingPassDepth : REAL; (* mm, finishing pass depth *)
    depthAdjAngle : LREAL; (* degrees, arc over which cut depth is adjusted. LREAL for position compatibility *)
    cutOverrunAngle : LREAL; (* degrees, arc len to overrun the last pass. LREAL for position compatibility *)
    EndOfCutProfile : BOOL := FALSE;
    feedRate : REAL; (* mm/sec, feed rate *)
    retractRate : REAL; (* deg/sec, velocity used when retracting the cutters *)
    accel : REAL;
    decel : REAL;
    setZeroOffset : REAL := 0.0; (* degrees. Offset applied when set zero is requested. *)
    depthMod : REAL := 0.0; (* mm, adjusment to the calculated finished depth *)
    offsetLimitPositive : LREAL; (* positive offset angle limit *)
    offsetLimitNegative : LREAL; (* negative offset angle limit *)

  END_STRUCT;

  sWp_Spindle :	STRUCT
    nomRpm : REAL; (* RPM, nominal *)
    accel : REAL;
    decel : REAL;
  END_STRUCT;

  sWp_ZAxis :	STRUCT
    indexSpeed : REAL; (* mm/sec *)
    accel : REAL;
    decel : REAL;
    indexDist : LREAL; (* mm. Index distance *)
    setZeroOffset : LREAL := 0.0; (* degrees. Offset applied when set zero is requested. *)
    zMod : LREAL := 0.0; (* mm, adjustment to Z position *)
    startOfCutPos : LREAL; (* position corresponding to index #1 -- start of cutting *)
    loadUnloadPos : LREAL; (* position to load/unload *)
  END_STRUCT;

  sWp_CfVfd :	STRUCT
    isInPressureControl : BOOL; (* H: Pressure ctrl, L: Speed Control *)
    runSpeedManualCtrl : REAL; (* rpm, manual run speed *)
    pressureSpAutoCtrl : REAL; (* psi, auto pressure setpoint *)
    accel : REAL;
    decel : REAL;
    eocCutoutWaitTime : TIME; (* how long to wait while idle at the end of a cycle before shutting off the cutting fluid *)
  END_STRUCT;

  sWp_PartDfn :	STRUCT  (* a part definition, but not a specific part *)
    number : STRING[15]; (* Part Number *)
    name : STRING[40]; (* Part Name *)
    nomId : REAL; (* mm, nominal inside diameter *)
    nomCutLength : LREAL; (* mm. Nominal length that cuts are made over. LREAL to be compatible with motion system *)
  END_STRUCT;

  sWp_Configuration : STRUCT
    name : STRING[40]; (* Config Name *)
    (* partDfn : sWp_PartDfn;  Part Definition *)
    cuttingHead : sWp_CuttingHead;
    spindle : sWp_Spindle;
    zAxis : sWp_ZAxis;
    cfVfd : sWp_CfVfd;
  END_STRUCT;

  (****************************************)
  (***** Hardware related structures  *****)
  (****************************************)

  sRioModuleHealth : STRUCT
    Slot01ModuleOk : BOOL;
    Slot02ModuleOk : BOOL;
    Slot03ModuleOk : BOOL;
    Slot04ModuleOk : BOOL;
    Slot05ModuleOk : BOOL;
    Slot06ModuleOk : BOOL;
    Slot07ModuleOk : BOOL;
    Slot08ModuleOk : BOOL;
    Slot09ModuleOk : BOOL;
    Slot10ModuleOk : BOOL;
    Slot11ModuleOk : BOOL;
    Slot12ModuleOk : BOOL;
    Slot13ModuleOk : BOOL;
    Slot14ModuleOk : BOOL;
    Slot15ModuleOk : BOOL;
    Slot16ModuleOk : BOOL;
    Slot17ModuleOk : BOOL;
    Slot18ModuleOk : BOOL;
    Slot19ModuleOk : BOOL;
    Slot20ModuleOk : BOOL;
    Slot21ModuleOk : BOOL;
    Slot22ModuleOk : BOOL;
    Slot23ModuleOk : BOOL;
    Slot24ModuleOk : BOOL;
    Slot25ModuleOk : BOOL;
    Slot26ModuleOk : BOOL;
    Slot27ModuleOk : BOOL;
    Slot28ModuleOk : BOOL;
    Slot29ModuleOk : BOOL;
    Slot30ModuleOk : BOOL;
    Slot31ModuleOk : BOOL;
    Slot32ModuleOk : BOOL;
  END_STRUCT;

END_TYPE
```

### Global.var
```iecst
VAR CONSTANT
  INVALID_SENTINEL : DINT:= -9999;
  INVALID_SENTINEL_REAL : REAL:= -9999.0;
  INVALID_SENTINEL_LREAL : LREAL:= -9999.0;

  (* Axis count is set here rather than in PlcLogic so it can be used to define arrays *)
  AXIS_COUNT : DINT := 8;

END_VAR

VAR RETAIN

  (* Retained and here in global so they can be permanent variables *)

  (* Tables used to lookup inner eccentric offset angles given a depth.
  50 element max, per lookup table, so break the lookup into pieces. *)
	gr_depthToAngleLu : sDepthToAngleLu;

  (* Part and Machine cfg *)
  gr_CfgCurrent : sWp_Configuration;
  gr_PartCurrent :sWp_Part;
  gr_CfgSaved : ARRAY[0..19] OF sWp_Configuration;
  gr_PartSaved : ARRAY[0..19] OF sWp_Part;

  (* Axis restore positions *)
  gr_AxSpindleRestorePos : McAcpAxRestorePosType;
  gr_AxOutERestorePos : McAcpAxRestorePosType;
  gr_AxInERestorePos : McAcpAxRestorePosType;
  gr_AxZRestorePos : McAcpAxRestorePosType;

  (* axis travel limits *)
  (* Set here in global so this can be made permanent *)
  gr_AxisPositionLimits : ARRAY[0..AXIS_COUNT] OF sMot_PositionLimits;

  (* analog input params *)
  gr_AI_FT_CFFlow_Params : sAnalogInputParams;
  gr_AI_LT_CFTankLevel_Params : sAnalogInputParams;
  gr_AI_PT_CFPumpOutlet_Params : sAnalogInputParams;
  gr_AI_PT_CFFilterOutlet_Params : sAnalogInputParams;
  gr_AI_DP_CFFilter_Params : sAnalogInputParams; (* virtual input derrived from 2 PTs *)

  (* digital input params *)
  gr_DI_LSL_CFTank_Params : sDigitalInputParams;
  gr_DI_ZS_CFTankLocator_Params : sDigitalInputParams;
  gr_DI_JI_480VACOk_Params : sDigitalInputParams;

END_VAR

VAR

END_VAR
```

### Library Logical/Libraries/GAProcIO (Iec) - Scale Analog functions

#### GAProcIO.typ
```iecst
(********************************************************************
 * COPYRIGHT -- General Atomics
 ********************************************************************
 * Library: GAProcIO
 * File: GAProcIO.typ
 * Author: Administrator
 * Created: September 11, 2015
 ********************************************************************
 * Data types of library GAProcIO
 ********************************************************************)

TYPE
	eGAPIO_RAW_SCALE_TYPE :
		(
		GAPIO_RWST_OFF := 0, (* do not process the chanel *)
		GAPIO_RWST_USINT := 1,
		GAPIO_RWST_SINT := 2,
		GAPIO_RWST_UINT := 3,
		GAPIO_RWST_INT := 4,
		GAPIO_RWST_UDINT := 5,
		GAPIO_RWST_DINT := 6,
    GAPIO_RWST_REAL := 7 (* LREAL not suppoeted by scaling routine *)
    (* RWST_LREAL := 8 *)
  ) := GAPIO_RWST_INT; (* default to int, since this is what most AIs are *)

  eGAPIO_PB_BEHAVIOR_TYPE :
    (
    GAPIO_PBBT_DISABLED   := 0, (* always off *)
    GAPIO_PBBT_MOMENTARY  := 1, (* active while pressed *)
    GAPIO_PBBT_OS_ON      := 2, (* oneshot on. Needs rising edge to turn on for 1 scan *)
    GAPIO_PBBT_PRESS_ON   := 3, (* press to turn on *)
    GAPIO_PBBT_PULSE_ON   := 4, (* turn on for a pulse *)
    GAPIO_PBBT_PRESS_OFF  := 5, (* press to turn off *)
    GAPIO_PBBT_TOGGLE     := 6  (* press to toggle *)
  ) := GAPIO_PBBT_MOMENTARY;

  sAnalogInput : 	STRUCT  (* 32 byte structure *)
    ModuleOk : BOOL; (* byte 0 H=okay *)
    ChannelOk : BOOL; (* byte 1 H=okay *)
    InRawUSINT : USINT; (* byte 2 *)
    InRawSINT : SINT; (* byte 3 *)
    InRawUINT : UINT; (* bytes 4-5 *)
    InRawINT : INT; (* bytes 6-7 *)
    InRawUDINT : UDINT; (* bytes 8-11 *)
    InRawDINT : DINT; (* bytes 12-15 *)
    InRawREAL : REAL; (* bytes 16-19 *)
    InScaled : REAL; (* byte 20-23 *)
    InScaledFiltered : REAL; (* byte 24-27 *)
    (* alarms *)
    (* bit packed integer - used so non-zero value means at least one alarm is active *)
    alms : UDINT := 0; (* b0:LoRange,b1:HiRange,b2:LoLoAlm,b3:LoAlm,b4:HiAlm,b5:HiHiAlm,b31:chErr *)
  END_STRUCT;

	sAnalogInputParams : 	STRUCT  (* analog scaling and alarm parameters *) (* raw scale type - how to interpret InRawBuffer *)
    CalcEUExternally : BOOL := FALSE; (* InScaled value is calculated outside the fbSclAlmAI fb *)
		LpEnable : BOOL := FALSE; (* turn off Low Pass Filter by default *)
		LpPreserveUnfiltered : BOOL := TRUE; (* F: filtered => unfiltered, T: keep separate *)
		AlmEnable : BOOL := FALSE;
		AlmLoLoEnable : BOOL := FALSE;
		AlmLoEnable : BOOL := FALSE;
		AlmHiEnable : BOOL := FALSE;
		AlmHiHiEnable : BOOL := FALSE; (* alarm thresholds - compare to EU (scaled) values *) (* disable range check and alarm thresholds by default if not specified *)
		RawType : eGAPIO_RAW_SCALE_TYPE := GAPIO_RWST_INT; (* default to int, since this is what most AIs are *) (* scaling parameters *)
		RawMin : REAL := 0.0; (* scale to 15 bits if not specified - a common value for ai modules *)
		RawMax : REAL := 32767.0;
		EuMin : REAL := 0.0; (* scale to percent if not specified *)
		EuMax : REAL := 100.0;
		RawOffset : REAL := 0.0; (* +/- counts value added to the raw value before scaling *)
		EuOffset : REAL := 0.0; (* +/- EU value added to EU after scaling *) (* Low Pass (Noise) filter parameters *)
		LpCoeff : REAL := 0.0; (* >=0 and <1. 0= no filtering. 0.99999= heavy filtering. *) (* alarm enables *) (* turn on or off all alarming except for out of range alarms *)
		AlmRangeThreshLo : REAL := -1.0E9;
		AlmRangeThreshHi : REAL := 1.0E9;
		AlmThreshLoLo : REAL := -1.0E9;
		AlmThreshLo : REAL := -1.0E9;
		AlmThreshHi : REAL := 1.0E9;
		AlmThreshHiHi : REAL := 1.0E9; (* alarm deadbands *) (* in % of range EU range *) (* use 0 to disable *)
		AlmDbLoPct : REAL := 1.0; (* pvs must rise above threshold by the corresponding value in order to be considered clear *)
		AlmDbHiPct : REAL := 1.0; (* pvs must drop below threshold by the corresponding value in order to be considered clear *) (* alarm time delays *) (* use 0 time to disable *)
		AlmLoOnDlyTime : TIME := T#1s;
		AlmHiOnDlyTime : TIME := T#1s; (* alarm off delay time - condition must clear for this long before being considered "gone" *)
		AlmLoOffDlyTime : TIME := T#1s;
		AlmHiOffDlyTime : TIME := T#1s;
  END_STRUCT;

  sDigitalInput : 	STRUCT
    ModuleOk : BOOL; (* H=okay *)
    ChannelOk : BOOL; (* H=okay *)
    InRaw : BOOL; (* raw input signal *)
    Value : BOOL; (* conditioned value *)
    spareBytes5_7 : ARRAY[5..7]OF BYTE;
    (* alarms *)
    (* bit packed integer - used so non-zero value means at least one alarm is active *)
    alms : UDINT := 0; (* b3:LoAlm,b4:HiAlm,b31:ch err,b0-2:reserved,b5-30:reserved *)
  END_STRUCT;

  sDigitalInputParams : 	STRUCT  (* digital signal processing and alarm parameters *)
    Enable : BOOL; (* H=process *)
    AlmEnable : BOOL := FALSE; (* set to process alarm *)
		AlmLoEnable : BOOL := FALSE; (* set to enable alarm if value is low *)
		AlmHiEnable : BOOL := FALSE; (* set to enable alarm if value is high *)
		Invert : BOOL := FALSE;
		OnDlyTime : TIME := T#0ms; (* delay time for value turning on *)
		OffDlyTime : TIME := T#0ms; (* delay time for value turning off *)
		AlmLoOnDlyTime : TIME := T#1s;
		AlmHiOnDlyTime : TIME := T#1s;
		AlmLoOffDlyTime : TIME := T#1s;
		AlmHiOffDlyTime : TIME := T#1s;
  END_STRUCT;

END_TYPE
```

#### GAProcIO.var
```iecst
(********************************************************************
 * COPYRIGHT -- General Atomics
 ********************************************************************
 * Library: GAScale
 * File: GAScale.var
 * Author: Administrator
 * Created: September 11, 2015
 ********************************************************************
 * Constants of library GAScale
 ********************************************************************)

VAR CONSTANT
  (* Use constants rather than enum so this isn't a DINT *)
  (* and is the same UDINT type as the alm registers. *)
  GAPIO_ALARM_NONE : UDINT      := 16#0000;
  GAPIO_ALARM_RANGELO : UDINT   := 16#0001; (* b0 *)
  GAPIO_ALARM_RANGEHI : UDINT   := 16#0002; (* b1 *)
  GAPIO_ALARM_LOLO : UDINT      := 16#0004; (* b2 *)
	GAPIO_ALARM_LO : UDINT        := 16#0008; (* b3 *)
	GAPIO_ALARM_HI : UDINT        := 16#0010; (* b4 *)
	GAPIO_ALARM_HIHI : UDINT      := 16#0020; (* b5 *)
	GAPIO_ALARM_CHANNEL : UDINT   := 16#80000000; (* b31 *)

END_VAR
```
